   1:  PR[GP1:91,2] = PR[GP1:90,2] + 36.838;
   1:L PR[91] R[100]mm/sec CNT100;
   1:  PR[GP1:91,1] = PR[GP1:90,1] + -37.461;
   1:  PR[GP1:91,2] = PR[GP1:90,2] + 32.882;
   1:L PR[91] R[100]mm/sec CNT100;
   1:  PR[GP1:91,1] = PR[GP1:90,1] + -42.341;
   1:  PR[GP1:91,2] = PR[GP1:90,2] + 27.004;
   1:L PR[91] R[100]mm/sec CNT100;
   1:  PR[GP1:91,1] = PR[GP1:90,1] + -45.904;
   1:  PR[GP1:91,2] = PR[GP1:90,2] + 21.052;
   1:L PR[91] R[100]mm/sec CNT100;
   1:  PR[GP1:91,1] = PR[GP1:90,1] + -48.927;
   1:  PR[GP1:91,2] = PR[GP1:90,2] + 14.203;
   1:L PR[91] R[100]mm/sec CNT100;
   1:  PR[GP1:91,1] = PR[GP1:90,1] + -50.193;
   1:  PR[GP1:91,2] = PR[GP1:90,2] + 7.261;
   1:L PR[91] R[100]mm/sec CNT100;
   1:  PR[GP1:91,1] = PR[GP1:90,1] + -51.214;
   1:  PR[GP1:91,2] = PR[GP1:90,2] + -0.059;
   1:L PR[91] R[100]mm/sec CNT100;
   1:  PR[GP1:91,1] = PR[GP1:90,1] + -49.961;
   1:  PR[GP1:91,2] = PR[GP1:90,2] + -6.907;
   1:L PR[91] R[100]mm/sec CNT100;
   1:  PR[GP1:91,1] = PR[GP1:90,1] + -48.922;
   1:  PR[GP1:91,2] = PR[GP1:90,2] + -14.358;
   1:L PR[91] R[100]mm/sec CNT100;
   1:  PR[GP1:91,1] = PR[GP1:90,1] + -45.904;
   1:  PR[GP1:91,2] = PR[GP1:90,2] + -21.195;
   1:L PR[91] R[100]mm/sec CNT100;
   1:  PR[GP1:91,1] = PR[GP1:90,1] + -42.341;
   1:  PR[GP1:91,2] = PR[GP1:90,2] + -27.147;
   1:L PR[91] R[100]mm/sec CNT100;
   1:  PR[GP1:91,1] = PR[GP1:90,1] + -37.450;
   1:  PR[GP1:91,2] = PR[GP1:90,2] + -33.039;
   1:L PR[91] R[100]mm/sec CNT100;
   1:  PR[GP1:91,1] = PR[GP1:90,1] + -32.224;
   1:  PR[GP1:91,2] = PR[GP1:90,2] + -37.231;
   1:L PR[91] R[100]mm/sec CNT100;
   1:  PR[GP1:91,1] = PR[GP1:90,1] + -26.484;
   1:  PR[GP1:91,2] = PR[GP1:90,2] + -41.295;
   1:L PR[91] R[100]mm/sec CNT100;
   1:  PR[GP1:91,1] = PR[GP1:90,1] + -19.923;
   1:  PR[GP1:91,2] = PR[GP1:90,2] + -43.838;
   1:L PR[91] R[100]mm/sec CNT100;
   1:  PR[GP1:91,1] = PR[GP1:90,1] + -13.684;
   1:  PR[GP1:91,2] = PR[GP1:90,2] + -45.938;
   1:L PR[91] R[100]mm/sec CNT100;
   1:  PR[GP1:91,1] = PR[GP1:90,1] + -6.476;
   1:  PR[GP1:91,2] = PR[GP1:90,2] + -46.831;
   1:L PR[91] R[100]mm/sec CNT100;
   1:  PR[GP1:91,1] = PR[GP1:90,1] + -0.261;
   1:  PR[GP1:91,2] = PR[GP1:90,2] + -46.697;
   1:L PR[91] R[100]mm/sec CNT100;
   1:  PR[GP1:91,1] = PR[GP1:90,1] + 0.472;
   1:  PR[GP1:91,2] = PR[GP1:90,2] + -46.698;
   1:L PR[91] R[100]mm/sec CNT100;
   1:  PR[GP1:91,1] = PR[GP1:90,1] + 6.688;
   1:  PR[GP1:91,2] = PR[GP1:90,2] + -46.831;
   1:L PR[91] R[100]mm/sec CNT100;
   1:  PR[GP1:91,1] = PR[GP1:90,1] + 13.897;
   1:  PR[GP1:91,2] = PR[GP1:90,2] + -45.938;
   1:L PR[91] R[100]mm/sec CNT100;
   1:  PR[GP1:91,1] = PR[GP1:90,1] + 20.136;
   1:  PR[GP1:91,2] = PR[GP1:90,2] + -43.838;
   1:L PR[91] R[100]mm/sec CNT100;
   1:  PR[GP1:91,1] = PR[GP1:90,1] + 26.682;
   1:  PR[GP1:91,2] = PR[GP1:90,2] + -41.301;
   1:L PR[91] R[100]mm/sec CNT100;
   1:  PR[GP1:91,1] = PR[GP1:90,1] + 32.087;
   1:  PR[GP1:91,2] = PR[GP1:90,2] + -36.981;
   1:L PR[91] R[100]mm/sec CNT100;
   1:  PR[GP1:91,1] = PR[GP1:90,1] + 37.676;
   1:  PR[GP1:91,2] = PR[GP1:90,2] + -33.023;
   1:L PR[91] R[100]mm/sec CNT100;
   1:  PR[GP1:91,1] = PR[GP1:90,1] + 42.555;
   1:  PR[GP1:91,2] = PR[GP1:90,2] + -27.145;
   1:L PR[91] R[100]mm/sec CNT100;
   1:  PR[GP1:91,1] = PR[GP1:90,1] + 46.117;
   1:  PR[GP1:91,2] = PR[GP1:90,2] + -21.197;
   1:L PR[91] R[100]mm/sec CNT100;
   1:  PR[GP1:91,1] = PR[GP1:90,1] + 49.141;
   1:  PR[GP1:91,2] = PR[GP1:90,2] + -14.349;
   1:L PR[91] R[100]mm/sec CNT100;
   1:  PR[GP1:91,1] = PR[GP1:90,1] + 50.406;
   1:  PR[GP1:91,2] = PR[GP1:90,2] + -7.404;
   1:L PR[91] R[100]mm/sec CNT100;
   1:  PR[GP1:91,1] = PR[GP1:90,1] + 51.427;
   1:  PR[GP1:91,2] = PR[GP1:90,2] + -0.085;
   1:L PR[91] R[100]mm/sec CNT100;
   1:  PR[GP1:91,1] = PR[GP1:90,1] + 50.175;
   1:  PR[GP1:91,2] = PR[GP1:90,2] + 6.766;
   1:L PR[91] R[100]mm/sec CNT100;
   1:  PR[GP1:91,1] = PR[GP1:90,1] + 49.135;
   1:  PR[GP1:91,2] = PR[GP1:90,2] + 14.217;
   1:L PR[91] R[100]mm/sec CNT100;
   1:  PR[GP1:91,1] = PR[GP1:90,1] + 46.117;
   1:  PR[GP1:91,2] = PR[GP1:90,2] + 21.053;
   1:L PR[91] R[100]mm/sec CNT100;
   1:  PR[GP1:91,1] = PR[GP1:90,1] + 42.555;
   1:  PR[GP1:91,2] = PR[GP1:90,2] + 27.002;
   1:L PR[91] R[100]mm/sec CNT100;
   1:  PR[GP1:91,1] = PR[GP1:90,1] + 37.664;
   1:  PR[GP1:91,2] = PR[GP1:90,2] + 32.894;
   1:L PR[91] R[100]mm/sec CNT100;
   1:  PR[GP1:91,1] = PR[GP1:90,1] + 32.438;
   1:  PR[GP1:91,2] = PR[GP1:90,2] + 37.087;
   1:L PR[91] R[100]mm/sec CNT100;
   1:  PR[GP1:91,1] = PR[GP1:90,1] + 26.697;
   1:  PR[GP1:91,2] = PR[GP1:90,2] + 41.152;
   1:L PR[91] R[100]mm/sec CNT100;
   1:  PR[GP1:91,1] = PR[GP1:90,1] + 20.134;
   1:  PR[GP1:91,2] = PR[GP1:90,2] + 43.695;
   1:L PR[91] R[100]mm/sec CNT100;
   1:  PR[GP1:91,1] = PR[GP1:90,1] + 13.896;
   1:  PR[GP1:91,2] = PR[GP1:90,2] + 45.794;
   1:L PR[91] R[100]mm/sec CNT100;
   1:  PR[GP1:91,1] = PR[GP1:90,1] + 6.686;
   1:  PR[GP1:91,2] = PR[GP1:90,2] + 46.687;
   1:L PR[91] R[100]mm/sec CNT100;
   1:  PR[GP1:91,1] = PR[GP1:90,1] + 0.472;
   1:  PR[GP1:91,2] = PR[GP1:90,2] + 46.554;
   1:L PR[91] R[100]mm/sec CNT100;
   1:  ! -- Layer/Ebene 193 -- !;
   1:  PR[91] = PR[90];
   1:  PR[GP1:91,1] = PR[GP1:90,1] + -0.240;
   1:  PR[GP1:91,2] = PR[GP1:90,2] + 46.709;
   1:  PR[GP1:91,3] = PR[GP1:90,3] + 118.035;
   1:L PR[91] R[100]mm/sec CNT100;
   1:  PR[GP1:91,1] = PR[GP1:90,1] + -6.104;
   1:  PR[GP1:91,2] = PR[GP1:90,2] + 46.835;
   1:L PR[91] R[100]mm/sec CNT100;
   1:  PR[GP1:91,1] = PR[GP1:90,1] + -13.586;
   1:  PR[GP1:91,2] = PR[GP1:90,2] + 45.908;
   1:L PR[91] R[100]mm/sec CNT100;
   1:  PR[GP1:91,1] = PR[GP1:90,1] + -19.471;
   1:  PR[GP1:91,2] = PR[GP1:90,2] + 43.928;
   1:L PR[91] R[100]mm/sec CNT100;
   1:  PR[GP1:91,1] = PR[GP1:90,1] + -26.286;
   1:  PR[GP1:91,2] = PR[GP1:90,2] + 41.286;
   1:L PR[91] R[100]mm/sec CNT100;
   1:  PR[GP1:91,1] = PR[GP1:90,1] + -31.386;
   1:  PR[GP1:91,2] = PR[GP1:90,2] + 37.212;
   1:L PR[91] R[100]mm/sec CNT100;
   1:  PR[GP1:91,1] = PR[GP1:90,1] + -37.220;
   1:  PR[GP1:91,2] = PR[GP1:90,2] + 33.081;
   1:L PR[91] R[100]mm/sec CNT100;
   1:  PR[GP1:91,1] = PR[GP1:90,1] + -42.317;
   1:  PR[GP1:91,2] = PR[GP1:90,2] + 26.942;
   1:L PR[91] R[100]mm/sec CNT100;
   1:  PR[GP1:91,1] = PR[GP1:90,1] + -45.678;
   1:  PR[GP1:91,2] = PR[GP1:90,2] + 21.327;
   1:L PR[91] R[100]mm/sec CNT100;
   1:  PR[GP1:91,1] = PR[GP1:90,1] + -48.842;
   1:  PR[GP1:91,2] = PR[GP1:90,2] + 14.160;
   1:L PR[91] R[100]mm/sec CNT100;
   1:  PR[GP1:91,1] = PR[GP1:90,1] + -50.036;
   1:  PR[GP1:91,2] = PR[GP1:90,2] + 7.611;
   1:L PR[91] R[100]mm/sec CNT100;
   1:  PR[GP1:91,1] = PR[GP1:90,1] + -51.106;
   1:  PR[GP1:91,2] = PR[GP1:90,2] + -0.059;
   1:L PR[91] R[100]mm/sec CNT100;
   1:  PR[GP1:91,1] = PR[GP1:90,1] + -49.924;
   1:  PR[GP1:91,2] = PR[GP1:90,2] + -6.518;
   1:L PR[91] R[100]mm/sec CNT100;
   1:  PR[GP1:91,1] = PR[GP1:90,1] + -48.837;
   1:  PR[GP1:91,2] = PR[GP1:90,2] + -14.315;
   1:L PR[91] R[100]mm/sec CNT100;
   1:  PR[GP1:91,1] = PR[GP1:90,1] + -45.678;
   1:  PR[GP1:91,2] = PR[GP1:90,2] + -21.471;
   1:L PR[91] R[100]mm/sec CNT100;
   1:  PR[GP1:91,1] = PR[GP1:90,1] + -42.317;
   1:  PR[GP1:91,2] = PR[GP1:90,2] + -27.085;
   1:L PR[91] R[100]mm/sec CNT100;
   1:  PR[GP1:91,1] = PR[GP1:90,1] + -37.209;
   1:  PR[GP1:91,2] = PR[GP1:90,2] + -33.238;
   1:L PR[91] R[100]mm/sec CNT100;
   1:  PR[GP1:91,1] = PR[GP1:90,1] + -32.280;
   1:  PR[GP1:91,2] = PR[GP1:90,2] + -37.192;
   1:L PR[91] R[100]mm/sec CNT100;
   1:  PR[GP1:91,1] = PR[GP1:90,1] + -26.304;
   1:  PR[GP1:91,2] = PR[GP1:90,2] + -41.423;
   1:L PR[91] R[100]mm/sec CNT100;
   1:  PR[GP1:91,1] = PR[GP1:90,1] + -19.472;
   1:  PR[GP1:91,2] = PR[GP1:90,2] + -44.071;
   1:L PR[91] R[100]mm/sec CNT100;
   1:  PR[GP1:91,1] = PR[GP1:90,1] + -13.588;
   1:  PR[GP1:91,2] = PR[GP1:90,2] + -46.052;
   1:L PR[91] R[100]mm/sec CNT100;
   1:  PR[GP1:91,1] = PR[GP1:90,1] + -6.105;
   1:  PR[GP1:91,2] = PR[GP1:90,2] + -46.979;
   1:L PR[91] R[100]mm/sec CNT100;
   1:  PR[GP1:91,1] = PR[GP1:90,1] + -0.241;
   1:  PR[GP1:91,2] = PR[GP1:90,2] + -46.853;
   1:L PR[91] R[100]mm/sec CNT100;
   1:  PR[GP1:91,1] = PR[GP1:90,1] + 0.452;
   1:L PR[91] R[100]mm/sec CNT100;
   1:  PR[GP1:91,1] = PR[GP1:90,1] + 6.317;
   1:  PR[GP1:91,2] = PR[GP1:90,2] + -46.979;
   1:L PR[91] R[100]mm/sec CNT100;
   1:  PR[GP1:91,1] = PR[GP1:90,1] + 13.801;
   1:  PR[GP1:91,2] = PR[GP1:90,2] + -46.052;
   1:L PR[91] R[100]mm/sec CNT100;
   1:  PR[GP1:91,1] = PR[GP1:90,1] + 19.685;
   1:  PR[GP1:91,2] = PR[GP1:90,2] + -44.071;
   1:L PR[91] R[100]mm/sec CNT100;
   1:  PR[GP1:91,1] = PR[GP1:90,1] + 26.501;
   1:  PR[GP1:91,2] = PR[GP1:90,2] + -41.430;
   1:L PR[91] R[100]mm/sec CNT100;
   1:  PR[GP1:91,1] = PR[GP1:90,1] + 31.600;
   1:  PR[GP1:91,2] = PR[GP1:90,2] + -37.354;
   1:L PR[91] R[100]mm/sec CNT100;
   1:  PR[GP1:91,1] = PR[GP1:90,1] + 37.436;
   1:  PR[GP1:91,2] = PR[GP1:90,2] + -33.222;
   1:L PR[91] R[100]mm/sec CNT100;
   1:  PR[GP1:91,1] = PR[GP1:90,1] + 42.531;
   1:  PR[GP1:91,2] = PR[GP1:90,2] + -27.083;
   1:L PR[91] R[100]mm/sec CNT100;
   1:  PR[GP1:91,1] = PR[GP1:90,1] + 45.891;
   1:  PR[GP1:91,2] = PR[GP1:90,2] + -21.472;
   1:L PR[91] R[100]mm/sec CNT100;
   1:  PR[GP1:91,1] = PR[GP1:90,1] + 49.055;
   1:  PR[GP1:91,2] = PR[GP1:90,2] + -14.305;
   1:L PR[91] R[100]mm/sec CNT100;
   1:  PR[GP1:91,1] = PR[GP1:90,1] + 50.249;
   1:  PR[GP1:91,2] = PR[GP1:90,2] + -7.755;
   1:L PR[91] R[100]mm/sec CNT100;
   1:  PR[GP1:91,1] = PR[GP1:90,1] + 51.319;
   1:  PR[GP1:91,2] = PR[GP1:90,2] + -0.085;
   1:L PR[91] R[100]mm/sec CNT100;
   1:  PR[GP1:91,1] = PR[GP1:90,1] + 50.137;
   1:  PR[GP1:91,2] = PR[GP1:90,2] + 6.377;
   1:L PR[91] R[100]mm/sec CNT100;
   1:  PR[GP1:91,1] = PR[GP1:90,1] + 49.050;
   1:  PR[GP1:91,2] = PR[GP1:90,2] + 14.174;
   1:L PR[91] R[100]mm/sec CNT100;
   1:  PR[GP1:91,1] = PR[GP1:90,1] + 45.891;
   1:  PR[GP1:91,2] = PR[GP1:90,2] + 21.329;
   1:L PR[91] R[100]mm/sec CNT100;
   1:  PR[GP1:91,1] = PR[GP1:90,1] + 42.531;
   1:  PR[GP1:91,2] = PR[GP1:90,2] + 26.940;
   1:L PR[91] R[100]mm/sec CNT100;
   1:  PR[GP1:91,1] = PR[GP1:90,1] + 37.423;
   1:  PR[GP1:91,2] = PR[GP1:90,2] + 33.092;
   1:L PR[91] R[100]mm/sec CNT100;
   1:  PR[GP1:91,1] = PR[GP1:90,1] + 32.494;
   1:  PR[GP1:91,2] = PR[GP1:90,2] + 37.048;
   1:L PR[91] R[100]mm/sec CNT100;
   1:  PR[GP1:91,1] = PR[GP1:90,1] + 26.517;
   1:  PR[GP1:91,2] = PR[GP1:90,2] + 41.280;
   1:L PR[91] R[100]mm/sec CNT100;
   1:  PR[GP1:91,1] = PR[GP1:90,1] + 19.684;
   1:  PR[GP1:91,2] = PR[GP1:90,2] + 43.928;
   1:L PR[91] R[100]mm/sec CNT100;
   1:  PR[GP1:91,1] = PR[GP1:90,1] + 13.799;
   1:  PR[GP1:91,2] = PR[GP1:90,2] + 45.908;
   1:L PR[91] R[100]mm/sec CNT100;
   1:  PR[GP1:91,1] = PR[GP1:90,1] + 6.315;
   1:  PR[GP1:91,2] = PR[GP1:90,2] + 46.835;
   1:L PR[91] R[100]mm/sec CNT100;
   1:  PR[GP1:91,1] = PR[GP1:90,1] + 0.452;
   1:  PR[GP1:91,2] = PR[GP1:90,2] + 46.709;
   1:L PR[91] R[100]mm/sec CNT100;
   1:  ! -- Layer/Ebene 194 -- !;
   1:  PR[91] = PR[90];
   1:  PR[GP1:91,1] = PR[GP1:90,1] + -0.220;
   1:  PR[GP1:91,2] = PR[GP1:90,2] + 46.865;
   1:  PR[GP1:91,3] = PR[GP1:90,3] + 118.645;
   1:L PR[91] R[100]mm/sec CNT100;
   1:  PR[GP1:91,1] = PR[GP1:90,1] + -5.733;
   1:  PR[GP1:91,2] = PR[GP1:90,2] + 46.983;
   1:L PR[91] R[100]mm/sec CNT100;
   1:  PR[GP1:91,1] = PR[GP1:90,1] + -13.490;
   1:  PR[GP1:91,2] = PR[GP1:90,2] + 46.022;
   1:L PR[91] R[100]mm/sec CNT100;
   1:  PR[GP1:91,1] = PR[GP1:90,1] + -19.021;
   1:  PR[GP1:91,2] = PR[GP1:90,2] + 44.161;
   1:L PR[91] R[100]mm/sec CNT100;
   1:  PR[GP1:91,1] = PR[GP1:90,1] + -26.106;
   1:  PR[GP1:91,2] = PR[GP1:90,2] + 41.415;
   1:L PR[91] R[100]mm/sec CNT100;
   1:  PR[GP1:91,1] = PR[GP1:90,1] + -30.900;
   1:  PR[GP1:91,2] = PR[GP1:90,2] + 37.585;
   1:L PR[91] R[100]mm/sec CNT100;
   1:  PR[GP1:91,1] = PR[GP1:90,1] + -36.980;
   1:  PR[GP1:91,2] = PR[GP1:90,2] + 33.280;
   1:L PR[91] R[100]mm/sec CNT100;
   1:  PR[GP1:91,1] = PR[GP1:90,1] + -42.293;
   1:  PR[GP1:91,2] = PR[GP1:90,2] + 26.880;
   1:L PR[91] R[100]mm/sec CNT100;
   1:  PR[GP1:91,1] = PR[GP1:90,1] + -45.452;
   1:  PR[GP1:91,2] = PR[GP1:90,2] + 21.603;
   1:L PR[91] R[100]mm/sec CNT100;
   1:  PR[GP1:91,1] = PR[GP1:90,1] + -48.757;
   1:  PR[GP1:91,2] = PR[GP1:90,2] + 14.117;
   1:L PR[91] R[100]mm/sec CNT100;
   1:  PR[GP1:91,1] = PR[GP1:90,1] + -49.879;
   1:  PR[GP1:91,2] = PR[GP1:90,2] + 7.962;
   1:L PR[91] R[100]mm/sec CNT100;
   1:  PR[GP1:91,1] = PR[GP1:90,1] + -50.998;
   1:  PR[GP1:91,2] = PR[GP1:90,2] + -0.059;
   1:L PR[91] R[100]mm/sec CNT100;
   1:  PR[GP1:91,1] = PR[GP1:90,1] + -49.887;
   1:  PR[GP1:91,2] = PR[GP1:90,2] + -6.130;
   1:L PR[91] R[100]mm/sec CNT100;
   1:  PR[GP1:91,1] = PR[GP1:90,1] + -48.752;
   1:  PR[GP1:91,2] = PR[GP1:90,2] + -14.272;
   1:L PR[91] R[100]mm/sec CNT100;
   1:  PR[GP1:91,1] = PR[GP1:90,1] + -45.452;
   1:  PR[GP1:91,2] = PR[GP1:90,2] + -21.747;
   1:L PR[91] R[100]mm/sec CNT100;
   1:  PR[GP1:91,1] = PR[GP1:90,1] + -42.294;
   1:  PR[GP1:91,2] = PR[GP1:90,2] + -27.023;
   1:L PR[91] R[100]mm/sec CNT100;
   1:  PR[GP1:91,1] = PR[GP1:90,1] + -36.969;
   1:  PR[GP1:91,2] = PR[GP1:90,2] + -33.437;
   1:L PR[91] R[100]mm/sec CNT100;
   1:  PR[GP1:91,1] = PR[GP1:90,1] + -32.336;
   1:  PR[GP1:91,2] = PR[GP1:90,2] + -37.153;
   1:L PR[91] R[100]mm/sec CNT100;
   1:  PR[GP1:91,1] = PR[GP1:90,1] + -26.124;
   1:  PR[GP1:91,2] = PR[GP1:90,2] + -41.552;
   1:L PR[91] R[100]mm/sec CNT100;
   1:  PR[GP1:91,1] = PR[GP1:90,1] + -19.022;
   1:  PR[GP1:91,2] = PR[GP1:90,2] + -44.304;
   1:L PR[91] R[100]mm/sec CNT100;
   1:  PR[GP1:91,1] = PR[GP1:90,1] + -13.491;
   1:  PR[GP1:91,2] = PR[GP1:90,2] + -46.166;
   1:L PR[91] R[100]mm/sec CNT100;
   1:  PR[GP1:91,1] = PR[GP1:90,1] + -5.734;
   1:  PR[GP1:91,2] = PR[GP1:90,2] + -47.127;
   1:L PR[91] R[100]mm/sec CNT100;
   1:  PR[GP1:91,1] = PR[GP1:90,1] + -0.221;
   1:  PR[GP1:91,2] = PR[GP1:90,2] + -47.009;
   1:L PR[91] R[100]mm/sec CNT100;
   1:  PR[GP1:91,1] = PR[GP1:90,1] + 0.432;
   1:L PR[91] R[100]mm/sec CNT100;
   1:  PR[GP1:91,1] = PR[GP1:90,1] + 5.946;
   1:  PR[GP1:91,2] = PR[GP1:90,2] + -47.127;
   1:L PR[91] R[100]mm/sec CNT100;
   1:  PR[GP1:91,1] = PR[GP1:90,1] + 13.704;
   1:  PR[GP1:91,2] = PR[GP1:90,2] + -46.166;
   1:L PR[91] R[100]mm/sec CNT100;
   1:  PR[GP1:91,1] = PR[GP1:90,1] + 19.235;
   1:  PR[GP1:91,2] = PR[GP1:90,2] + -44.304;
   1:L PR[91] R[100]mm/sec CNT100;
   1:  PR[GP1:91,1] = PR[GP1:90,1] + 26.321;
   1:  PR[GP1:91,2] = PR[GP1:90,2] + -41.558;
   1:L PR[91] R[100]mm/sec CNT100;
   1:  PR[GP1:91,1] = PR[GP1:90,1] + 31.114;
   1:  PR[GP1:91,2] = PR[GP1:90,2] + -37.727;
   1:L PR[91] R[100]mm/sec CNT100;
   1:  PR[GP1:91,1] = PR[GP1:90,1] + 37.195;
   1:  PR[GP1:91,2] = PR[GP1:90,2] + -33.421;
   1:L PR[91] R[100]mm/sec CNT100;
   1:  PR[GP1:91,1] = PR[GP1:90,1] + 42.507;
   1:  PR[GP1:91,2] = PR[GP1:90,2] + -27.022;
   1:L PR[91] R[100]mm/sec CNT100;
   1:  PR[GP1:91,1] = PR[GP1:90,1] + 45.665;
   1:  PR[GP1:91,2] = PR[GP1:90,2] + -21.748;
   1:L PR[91] R[100]mm/sec CNT100;
   1:  PR[GP1:91,1] = PR[GP1:90,1] + 48.970;
   1:  PR[GP1:91,2] = PR[GP1:90,2] + -14.262;
   1:L PR[91] R[100]mm/sec CNT100;
   1:  PR[GP1:91,1] = PR[GP1:90,1] + 50.092;
   1:  PR[GP1:91,2] = PR[GP1:90,2] + -8.106;
   1:L PR[91] R[100]mm/sec CNT100;
   1:  PR[GP1:91,1] = PR[GP1:90,1] + 51.211;
   1:  PR[GP1:91,2] = PR[GP1:90,2] + -0.085;
   1:L PR[91] R[100]mm/sec CNT100;
   1:  PR[GP1:91,1] = PR[GP1:90,1] + 50.100;
   1:  PR[GP1:91,2] = PR[GP1:90,2] + 5.988;
   1:L PR[91] R[100]mm/sec CNT100;
   1:  PR[GP1:91,1] = PR[GP1:90,1] + 48.965;
   1:  PR[GP1:91,2] = PR[GP1:90,2] + 14.130;
   1:L PR[91] R[100]mm/sec CNT100;
   1:  PR[GP1:91,1] = PR[GP1:90,1] + 45.665;
   1:  PR[GP1:91,2] = PR[GP1:90,2] + 21.604;
   1:L PR[91] R[100]mm/sec CNT100;
   1:  PR[GP1:91,1] = PR[GP1:90,1] + 42.507;
   1:  PR[GP1:91,2] = PR[GP1:90,2] + 26.878;
   1:L PR[91] R[100]mm/sec CNT100;
   1:  PR[GP1:91,1] = PR[GP1:90,1] + 37.183;
   1:  PR[GP1:91,2] = PR[GP1:90,2] + 33.291;
   1:L PR[91] R[100]mm/sec CNT100;
   1:  PR[GP1:91,1] = PR[GP1:90,1] + 32.550;
   1:  PR[GP1:91,2] = PR[GP1:90,2] + 37.009;
   1:L PR[91] R[100]mm/sec CNT100;
   1:  PR[GP1:91,1] = PR[GP1:90,1] + 26.336;
   1:  PR[GP1:91,2] = PR[GP1:90,2] + 41.408;
   1:L PR[91] R[100]mm/sec CNT100;
   1:  PR[GP1:91,1] = PR[GP1:90,1] + 19.234;
   1:  PR[GP1:91,2] = PR[GP1:90,2] + 44.161;
   1:L PR[91] R[100]mm/sec CNT100;
   1:  PR[GP1:91,1] = PR[GP1:90,1] + 13.702;
   1:  PR[GP1:91,2] = PR[GP1:90,2] + 46.023;
   1:L PR[91] R[100]mm/sec CNT100;
   1:  PR[GP1:91,1] = PR[GP1:90,1] + 5.945;
   1:  PR[GP1:91,2] = PR[GP1:90,2] + 46.983;
   1:L PR[91] R[100]mm/sec CNT100;
   1:  PR[GP1:91,1] = PR[GP1:90,1] + 0.432;
   1:  PR[GP1:91,2] = PR[GP1:90,2] + 46.865;
   1:L PR[91] R[100]mm/sec CNT100;
   1:  ! -- Layer/Ebene 195 -- !;
   1:  PR[91] = PR[90];
   1:  PR[GP1:91,1] = PR[GP1:90,1] + -0.200;
   1:  PR[GP1:91,2] = PR[GP1:90,2] + 47.020;
   1:  PR[GP1:91,3] = PR[GP1:90,3] + 119.255;
   1:L PR[91] R[100]mm/sec CNT100;
   1:  PR[GP1:91,1] = PR[GP1:90,1] + -5.362;
   1:  PR[GP1:91,2] = PR[GP1:90,2] + 47.131;
   1:L PR[91] R[100]mm/sec CNT100;
   1:  PR[GP1:91,1] = PR[GP1:90,1] + -13.393;
   1:  PR[GP1:91,2] = PR[GP1:90,2] + 46.136;
   1:L PR[91] R[100]mm/sec CNT100;
   1:  PR[GP1:91,1] = PR[GP1:90,1] + -18.571;
   1:  PR[GP1:91,2] = PR[GP1:90,2] + 44.394;
   1:L PR[91] R[100]mm/sec CNT100;
   1:  PR[GP1:91,1] = PR[GP1:90,1] + -25.926;
   1:  PR[GP1:91,2] = PR[GP1:90,2] + 41.543;
   1:L PR[91] R[100]mm/sec CNT100;
   1:  PR[GP1:91,1] = PR[GP1:90,1] + -30.413;
   1:  PR[GP1:91,2] = PR[GP1:90,2] + 37.958;
   1:L PR[91] R[100]mm/sec CNT100;
   1:  PR[GP1:91,1] = PR[GP1:90,1] + -36.739;
   1:  PR[GP1:91,2] = PR[GP1:90,2] + 33.479;
   1:L PR[91] R[100]mm/sec CNT100;
   1:  PR[GP1:91,1] = PR[GP1:90,1] + -42.269;
   1:  PR[GP1:91,2] = PR[GP1:90,2] + 26.818;
   1:L PR[91] R[100]mm/sec CNT100;
   1:  PR[GP1:91,1] = PR[GP1:90,1] + -45.226;
   1:  PR[GP1:91,2] = PR[GP1:90,2] + 21.879;
   1:L PR[91] R[100]mm/sec CNT100;
   1:  PR[GP1:91,1] = PR[GP1:90,1] + -48.671;
   1:  PR[GP1:91,2] = PR[GP1:90,2] + 14.074;
   1:L PR[91] R[100]mm/sec CNT100;
   1:  PR[GP1:91,1] = PR[GP1:90,1] + -49.722;
   1:  PR[GP1:91,2] = PR[GP1:90,2] + 8.313;
   1:L PR[91] R[100]mm/sec CNT100;
   1:  PR[GP1:91,1] = PR[GP1:90,1] + -50.889;
   1:  PR[GP1:91,2] = PR[GP1:90,2] + -0.059;
   1:L PR[91] R[100]mm/sec CNT100;
   1:  PR[GP1:91,1] = PR[GP1:90,1] + -49.850;
   1:  PR[GP1:91,2] = PR[GP1:90,2] + -5.741;
   1:L PR[91] R[100]mm/sec CNT100;
   1:  PR[GP1:91,1] = PR[GP1:90,1] + -48.666;
   1:  PR[GP1:91,2] = PR[GP1:90,2] + -14.229;
   1:L PR[91] R[100]mm/sec CNT100;
   1:  PR[GP1:91,1] = PR[GP1:90,1] + -45.226;
   1:  PR[GP1:91,2] = PR[GP1:90,2] + -22.022;
   1:L PR[91] R[100]mm/sec CNT100;
   1:  PR[GP1:91,1] = PR[GP1:90,1] + -42.270;
   1:  PR[GP1:91,2] = PR[GP1:90,2] + -26.961;
   1:L PR[91] R[100]mm/sec CNT100;
   1:  PR[GP1:91,1] = PR[GP1:90,1] + -36.728;
   1:  PR[GP1:91,2] = PR[GP1:90,2] + -33.636;
   1:L PR[91] R[100]mm/sec CNT100;
   1:  PR[GP1:91,1] = PR[GP1:90,1] + -32.392;
   1:  PR[GP1:91,2] = PR[GP1:90,2] + -37.114;
   1:L PR[91] R[100]mm/sec CNT100;
   1:  PR[GP1:91,1] = PR[GP1:90,1] + -25.943;
   1:  PR[GP1:91,2] = PR[GP1:90,2] + -41.680;
   1:L PR[91] R[100]mm/sec CNT100;
   1:  PR[GP1:91,1] = PR[GP1:90,1] + -18.572;
   1:  PR[GP1:91,2] = PR[GP1:90,2] + -44.537;
   1:L PR[91] R[100]mm/sec CNT100;
   1:  PR[GP1:91,1] = PR[GP1:90,1] + -13.394;
   1:  PR[GP1:91,2] = PR[GP1:90,2] + -46.280;
   1:L PR[91] R[100]mm/sec CNT100;
   1:  PR[GP1:91,1] = PR[GP1:90,1] + -5.364;
   1:  PR[GP1:91,2] = PR[GP1:90,2] + -47.275;
   1:L PR[91] R[100]mm/sec CNT100;
   1:  PR[GP1:91,1] = PR[GP1:90,1] + -0.201;
   1:  PR[GP1:91,2] = PR[GP1:90,2] + -47.164;
   1:L PR[91] R[100]mm/sec CNT100;
   1:  PR[GP1:91,1] = PR[GP1:90,1] + 0.412;
   1:L PR[91] R[100]mm/sec CNT100;
   1:  PR[GP1:91,1] = PR[GP1:90,1] + 5.575;
   1:  PR[GP1:91,2] = PR[GP1:90,2] + -47.275;
   1:L PR[91] R[100]mm/sec CNT100;
   1:  PR[GP1:91,1] = PR[GP1:90,1] + 13.607;
   1:  PR[GP1:91,2] = PR[GP1:90,2] + -46.280;
   1:L PR[91] R[100]mm/sec CNT100;
   1:  PR[GP1:91,1] = PR[GP1:90,1] + 18.784;
   1:  PR[GP1:91,2] = PR[GP1:90,2] + -44.537;
   1:L PR[91] R[100]mm/sec CNT100;
   1:  PR[GP1:91,1] = PR[GP1:90,1] + 26.140;
   1:  PR[GP1:91,2] = PR[GP1:90,2] + -41.687;
   1:L PR[91] R[100]mm/sec CNT100;
   1:  PR[GP1:91,1] = PR[GP1:90,1] + 30.627;
   1:  PR[GP1:91,2] = PR[GP1:90,2] + -38.101;
   1:L PR[91] R[100]mm/sec CNT100;
   1:  PR[GP1:91,1] = PR[GP1:90,1] + 36.955;
   1:  PR[GP1:91,2] = PR[GP1:90,2] + -33.620;
   1:L PR[91] R[100]mm/sec CNT100;
   1:  PR[GP1:91,1] = PR[GP1:90,1] + 42.484;
   1:  PR[GP1:91,2] = PR[GP1:90,2] + -26.960;
   1:L PR[91] R[100]mm/sec CNT100;
   1:  PR[GP1:91,1] = PR[GP1:90,1] + 45.439;
   1:  PR[GP1:91,2] = PR[GP1:90,2] + -22.024;
   1:L PR[91] R[100]mm/sec CNT100;
   1:  PR[GP1:91,1] = PR[GP1:90,1] + 48.885;
   1:  PR[GP1:91,2] = PR[GP1:90,2] + -14.219;
   1:L PR[91] R[100]mm/sec CNT100;
   1:  PR[GP1:91,1] = PR[GP1:90,1] + 49.935;
   1:  PR[GP1:91,2] = PR[GP1:90,2] + -8.456;
   1:L PR[91] R[100]mm/sec CNT100;
   1:  PR[GP1:91,1] = PR[GP1:90,1] + 51.103;
   1:  PR[GP1:91,2] = PR[GP1:90,2] + -0.085;
   1:L PR[91] R[100]mm/sec CNT100;
   1:  PR[GP1:91,1] = PR[GP1:90,1] + 50.063;
   1:  PR[GP1:91,2] = PR[GP1:90,2] + 5.599;
   1:L PR[91] R[100]mm/sec CNT100;
   1:  PR[GP1:91,1] = PR[GP1:90,1] + 48.880;
   1:  PR[GP1:91,2] = PR[GP1:90,2] + 14.087;
   1:L PR[91] R[100]mm/sec CNT100;
   1:  PR[GP1:91,1] = PR[GP1:90,1] + 45.439;
   1:  PR[GP1:91,2] = PR[GP1:90,2] + 21.880;
   1:L PR[91] R[100]mm/sec CNT100;
   1:  PR[GP1:91,1] = PR[GP1:90,1] + 42.483;
   1:  PR[GP1:91,2] = PR[GP1:90,2] + 26.816;
   1:L PR[91] R[100]mm/sec CNT100;
   1:  PR[GP1:91,1] = PR[GP1:90,1] + 36.943;
   1:  PR[GP1:91,2] = PR[GP1:90,2] + 33.490;
   1:L PR[91] R[100]mm/sec CNT100;
   1:  PR[GP1:91,1] = PR[GP1:90,1] + 32.606;
   1:  PR[GP1:91,2] = PR[GP1:90,2] + 36.970;
   1:L PR[91] R[100]mm/sec CNT100;
   1:  PR[GP1:91,1] = PR[GP1:90,1] + 26.156;
   1:  PR[GP1:91,2] = PR[GP1:90,2] + 41.537;
   1:L PR[91] R[100]mm/sec CNT100;
   1:  PR[GP1:91,1] = PR[GP1:90,1] + 18.783;
   1:  PR[GP1:91,2] = PR[GP1:90,2] + 44.394;
   1:L PR[91] R[100]mm/sec CNT100;
   1:  PR[GP1:91,1] = PR[GP1:90,1] + 13.606;
   1:  PR[GP1:91,2] = PR[GP1:90,2] + 46.137;
   1:L PR[91] R[100]mm/sec CNT100;
   1:  PR[GP1:91,1] = PR[GP1:90,1] + 5.574;
   1:  PR[GP1:91,2] = PR[GP1:90,2] + 47.131;
   1:L PR[91] R[100]mm/sec CNT100;
   1:  PR[GP1:91,1] = PR[GP1:90,1] + 0.411;
   1:  PR[GP1:91,2] = PR[GP1:90,2] + 47.020;
   1:L PR[91] R[100]mm/sec CNT100;
   1:  ! -- Layer/Ebene 196 -- !;
   1:  PR[91] = PR[90];
   1:  PR[GP1:91,1] = PR[GP1:90,1] + -0.180;
   1:  PR[GP1:91,2] = PR[GP1:90,2] + 47.176;
   1:  PR[GP1:91,3] = PR[GP1:90,3] + 119.865;
   1:L PR[91] R[100]mm/sec CNT100;
   1:  PR[GP1:91,1] = PR[GP1:90,1] + -4.992;
   1:  PR[GP1:91,2] = PR[GP1:90,2] + 47.279;
   1:L PR[91] R[100]mm/sec CNT100;
   1:  PR[GP1:91,1] = PR[GP1:90,1] + -13.297;
   1:  PR[GP1:91,2] = PR[GP1:90,2] + 46.250;
   1:L PR[91] R[100]mm/sec CNT100;
   1:  PR[GP1:91,1] = PR[GP1:90,1] + -18.120;
   1:  PR[GP1:91,2] = PR[GP1:90,2] + 44.627;
   1:L PR[91] R[100]mm/sec CNT100;
   1:  PR[GP1:91,1] = PR[GP1:90,1] + -25.746;
   1:  PR[GP1:91,2] = PR[GP1:90,2] + 41.672;
   1:L PR[91] R[100]mm/sec CNT100;
   1:  PR[GP1:91,1] = PR[GP1:90,1] + -29.926;
   1:  PR[GP1:91,2] = PR[GP1:90,2] + 38.331;
   1:L PR[91] R[100]mm/sec CNT100;
   1:  PR[GP1:91,1] = PR[GP1:90,1] + -36.499;
   1:  PR[GP1:91,2] = PR[GP1:90,2] + 33.677;
   1:L PR[91] R[100]mm/sec CNT100;
   1:  PR[GP1:91,1] = PR[GP1:90,1] + -42.245;
   1:  PR[GP1:91,2] = PR[GP1:90,2] + 26.756;
   1:L PR[91] R[100]mm/sec CNT100;
   1:  PR[GP1:91,1] = PR[GP1:90,1] + -45.000;
   1:  PR[GP1:91,2] = PR[GP1:90,2] + 22.155;
   1:L PR[91] R[100]mm/sec CNT100;
   1:  PR[GP1:91,1] = PR[GP1:90,1] + -48.586;
   1:  PR[GP1:91,2] = PR[GP1:90,2] + 14.030;
   1:L PR[91] R[100]mm/sec CNT100;
   1:  PR[GP1:91,1] = PR[GP1:90,1] + -49.565;
   1:  PR[GP1:91,2] = PR[GP1:90,2] + 8.663;
   1:L PR[91] R[100]mm/sec CNT100;
   1:  PR[GP1:91,1] = PR[GP1:90,1] + -50.781;
   1:  PR[GP1:91,2] = PR[GP1:90,2] + -0.059;
   1:L PR[91] R[100]mm/sec CNT100;
   1:  PR[GP1:91,1] = PR[GP1:90,1] + -49.813;
   1:  PR[GP1:91,2] = PR[GP1:90,2] + -5.353;
   1:L PR[91] R[100]mm/sec CNT100;
   1:  PR[GP1:91,1] = PR[GP1:90,1] + -48.581;
   1:  PR[GP1:91,2] = PR[GP1:90,2] + -14.186;
   1:L PR[91] R[100]mm/sec CNT100;
   1:  PR[GP1:91,1] = PR[GP1:90,1] + -45.000;
   1:  PR[GP1:91,2] = PR[GP1:90,2] + -22.298;
   1:L PR[91] R[100]mm/sec CNT100;
   1:  PR[GP1:91,1] = PR[GP1:90,1] + -42.246;
   1:  PR[GP1:91,2] = PR[GP1:90,2] + -26.899;
   1:L PR[91] R[100]mm/sec CNT100;
   1:  PR[GP1:91,1] = PR[GP1:90,1] + -36.488;
   1:  PR[GP1:91,2] = PR[GP1:90,2] + -33.835;
   1:L PR[91] R[100]mm/sec CNT100;
   1:  PR[GP1:91,1] = PR[GP1:90,1] + -32.448;
   1:  PR[GP1:91,2] = PR[GP1:90,2] + -37.075;
   1:L PR[91] R[100]mm/sec CNT100;
   1:  PR[GP1:91,1] = PR[GP1:90,1] + -25.763;
   1:  PR[GP1:91,2] = PR[GP1:90,2] + -41.809;
   1:L PR[91] R[100]mm/sec CNT100;
   1:  PR[GP1:91,1] = PR[GP1:90,1] + -18.121;
   1:  PR[GP1:91,2] = PR[GP1:90,2] + -44.770;
   1:L PR[91] R[100]mm/sec CNT100;
   1:  PR[GP1:91,1] = PR[GP1:90,1] + -13.298;
   1:  PR[GP1:91,2] = PR[GP1:90,2] + -46.394;
   1:L PR[91] R[100]mm/sec CNT100;
   1:  PR[GP1:91,1] = PR[GP1:90,1] + -4.993;
   1:  PR[GP1:91,2] = PR[GP1:90,2] + -47.423;
   1:L PR[91] R[100]mm/sec CNT100;
   1:  PR[GP1:91,1] = PR[GP1:90,1] + -0.180;
   1:  PR[GP1:91,2] = PR[GP1:90,2] + -47.320;
   1:L PR[91] R[100]mm/sec CNT100;
   1:  PR[GP1:91,1] = PR[GP1:90,1] + 0.391;
   1:L PR[91] R[100]mm/sec CNT100;
   1:  PR[GP1:91,1] = PR[GP1:90,1] + 5.204;
   1:  PR[GP1:91,2] = PR[GP1:90,2] + -47.423;
   1:L PR[91] R[100]mm/sec CNT100;
   1:  PR[GP1:91,1] = PR[GP1:90,1] + 13.510;
   1:  PR[GP1:91,2] = PR[GP1:90,2] + -46.395;
   1:L PR[91] R[100]mm/sec CNT100;
   1:  PR[GP1:91,1] = PR[GP1:90,1] + 18.334;
   1:  PR[GP1:91,2] = PR[GP1:90,2] + -44.771;
   1:L PR[91] R[100]mm/sec CNT100;
   1:  PR[GP1:91,1] = PR[GP1:90,1] + 25.960;
   1:  PR[GP1:91,2] = PR[GP1:90,2] + -41.815;
   1:L PR[91] R[100]mm/sec CNT100;
   1:  PR[GP1:91,1] = PR[GP1:90,1] + 30.140;
   1:  PR[GP1:91,2] = PR[GP1:90,2] + -38.474;
   1:L PR[91] R[100]mm/sec CNT100;
   1:  PR[GP1:91,1] = PR[GP1:90,1] + 36.714;
   1:  PR[GP1:91,2] = PR[GP1:90,2] + -33.819;
   1:L PR[91] R[100]mm/sec CNT100;
   1:  PR[GP1:91,1] = PR[GP1:90,1] + 42.460;
   1:  PR[GP1:91,2] = PR[GP1:90,2] + -26.898;
   1:L PR[91] R[100]mm/sec CNT100;
   1:  PR[GP1:91,1] = PR[GP1:90,1] + 45.213;
   1:  PR[GP1:91,2] = PR[GP1:90,2] + -22.299;
   1:L PR[91] R[100]mm/sec CNT100;
   1:  PR[GP1:91,1] = PR[GP1:90,1] + 48.800;
   1:  PR[GP1:91,2] = PR[GP1:90,2] + -14.175;
   1:L PR[91] R[100]mm/sec CNT100;
   1:  PR[GP1:91,1] = PR[GP1:90,1] + 49.778;
   1:  PR[GP1:91,2] = PR[GP1:90,2] + -8.807;
   1:L PR[91] R[100]mm/sec CNT100;
   1:  PR[GP1:91,1] = PR[GP1:90,1] + 50.995;
   1:  PR[GP1:91,2] = PR[GP1:90,2] + -0.085;
   1:L PR[91] R[100]mm/sec CNT100;
   1:  PR[GP1:91,1] = PR[GP1:90,1] + 50.026;
   1:  PR[GP1:91,2] = PR[GP1:90,2] + 5.211;
   1:L PR[91] R[100]mm/sec CNT100;
   1:  PR[GP1:91,1] = PR[GP1:90,1] + 48.794;
   1:  PR[GP1:91,2] = PR[GP1:90,2] + 14.043;
   1:L PR[91] R[100]mm/sec CNT100;
   1:  PR[GP1:91,1] = PR[GP1:90,1] + 45.213;
   1:  PR[GP1:91,2] = PR[GP1:90,2] + 22.156;
   1:L PR[91] R[100]mm/sec CNT100;
   1:  PR[GP1:91,1] = PR[GP1:90,1] + 42.459;
   1:  PR[GP1:91,2] = PR[GP1:90,2] + 26.754;
   1:L PR[91] R[100]mm/sec CNT100;
   1:  PR[GP1:91,1] = PR[GP1:90,1] + 36.702;
   1:  PR[GP1:91,2] = PR[GP1:90,2] + 33.689;
   1:L PR[91] R[100]mm/sec CNT100;
   1:  PR[GP1:91,1] = PR[GP1:90,1] + 32.662;
   1:  PR[GP1:91,2] = PR[GP1:90,2] + 36.931;
   1:L PR[91] R[100]mm/sec CNT100;
   1:  PR[GP1:91,1] = PR[GP1:90,1] + 25.976;
   1:  PR[GP1:91,2] = PR[GP1:90,2] + 41.665;
   1:L PR[91] R[100]mm/sec CNT100;
   1:  PR[GP1:91,1] = PR[GP1:90,1] + 18.333;
   1:  PR[GP1:91,2] = PR[GP1:90,2] + 44.627;
   1:L PR[91] R[100]mm/sec CNT100;
   1:  PR[GP1:91,1] = PR[GP1:90,1] + 13.509;
   1:  PR[GP1:91,2] = PR[GP1:90,2] + 46.251;
   1:L PR[91] R[100]mm/sec CNT100;
   1:  PR[GP1:91,1] = PR[GP1:90,1] + 5.203;
   1:  PR[GP1:91,2] = PR[GP1:90,2] + 47.279;
   1:L PR[91] R[100]mm/sec CNT100;
   1:  PR[GP1:91,1] = PR[GP1:90,1] + 0.391;
   1:  PR[GP1:91,2] = PR[GP1:90,2] + 47.176;
   1:L PR[91] R[100]mm/sec CNT100;
   1:  ! -- Layer/Ebene 197 -- !;
   1:  PR[91] = PR[90];
   1:  PR[GP1:91,1] = PR[GP1:90,1] + -4.621;
   1:  PR[GP1:91,2] = PR[GP1:90,2] + 47.427;
   1:  PR[GP1:91,3] = PR[GP1:90,3] + 120.475;
   1:L PR[91] R[100]mm/sec CNT100;
   1:  PR[GP1:91,1] = PR[GP1:90,1] + -13.200;
   1:  PR[GP1:91,2] = PR[GP1:90,2] + 46.364;
   1:L PR[91] R[100]mm/sec CNT100;
   1:  PR[GP1:91,1] = PR[GP1:90,1] + -17.670;
   1:  PR[GP1:91,2] = PR[GP1:90,2] + 44.860;
   1:L PR[91] R[100]mm/sec CNT100;
   1:  PR[GP1:91,1] = PR[GP1:90,1] + -25.565;
   1:  PR[GP1:91,2] = PR[GP1:90,2] + 41.800;
   1:L PR[91] R[100]mm/sec CNT100;
   1:  PR[GP1:91,1] = PR[GP1:90,1] + -29.440;
   1:  PR[GP1:91,2] = PR[GP1:90,2] + 38.705;
   1:L PR[91] R[100]mm/sec CNT100;
   1:  PR[GP1:91,1] = PR[GP1:90,1] + -36.259;
   1:  PR[GP1:91,2] = PR[GP1:90,2] + 33.876;
   1:L PR[91] R[100]mm/sec CNT100;
   1:  PR[GP1:91,1] = PR[GP1:90,1] + -42.221;
   1:  PR[GP1:91,2] = PR[GP1:90,2] + 26.694;
   1:L PR[91] R[100]mm/sec CNT100;
   1:  PR[GP1:91,1] = PR[GP1:90,1] + -44.774;
   1:  PR[GP1:91,2] = PR[GP1:90,2] + 22.430;
   1:L PR[91] R[100]mm/sec CNT100;
   1:  PR[GP1:91,1] = PR[GP1:90,1] + -48.501;
   1:  PR[GP1:91,2] = PR[GP1:90,2] + 13.987;
   1:L PR[91] R[100]mm/sec CNT100;
   1:  PR[GP1:91,1] = PR[GP1:90,1] + -49.408;
   1:  PR[GP1:91,2] = PR[GP1:90,2] + 9.014;
   1:L PR[91] R[100]mm/sec CNT100;
   1:  PR[GP1:91,1] = PR[GP1:90,1] + -50.673;
   1:  PR[GP1:91,2] = PR[GP1:90,2] + -0.059;
   1:L PR[91] R[100]mm/sec CNT100;
   1:  PR[GP1:91,1] = PR[GP1:90,1] + -49.776;
   1:  PR[GP1:91,2] = PR[GP1:90,2] + -4.964;
   1:L PR[91] R[100]mm/sec CNT100;
   1:  PR[GP1:91,1] = PR[GP1:90,1] + -48.496;
   1:  PR[GP1:91,2] = PR[GP1:90,2] + -14.142;
   1:L PR[91] R[100]mm/sec CNT100;
   1:  PR[GP1:91,1] = PR[GP1:90,1] + -44.774;
   1:  PR[GP1:91,2] = PR[GP1:90,2] + -22.574;
   1:L PR[91] R[100]mm/sec CNT100;
   1:  PR[GP1:91,1] = PR[GP1:90,1] + -42.222;
   1:  PR[GP1:91,2] = PR[GP1:90,2] + -26.837;
   1:L PR[91] R[100]mm/sec CNT100;
   1:  PR[GP1:91,1] = PR[GP1:90,1] + -36.247;
   1:  PR[GP1:91,2] = PR[GP1:90,2] + -34.034;
   1:L PR[91] R[100]mm/sec CNT100;
   1:  PR[GP1:91,1] = PR[GP1:90,1] + -32.504;
   1:  PR[GP1:91,2] = PR[GP1:90,2] + -37.036;
   1:L PR[91] R[100]mm/sec CNT100;
   1:  PR[GP1:91,1] = PR[GP1:90,1] + -25.583;
   1:  PR[GP1:91,2] = PR[GP1:90,2] + -41.937;
   1:L PR[91] R[100]mm/sec CNT100;
   1:  PR[GP1:91,1] = PR[GP1:90,1] + -17.671;
   1:  PR[GP1:91,2] = PR[GP1:90,2] + -45.004;
   1:L PR[91] R[100]mm/sec CNT100;
   1:  PR[GP1:91,1] = PR[GP1:90,1] + -13.201;
   1:  PR[GP1:91,2] = PR[GP1:90,2] + -46.508;
   1:L PR[91] R[100]mm/sec CNT100;
   1:  PR[GP1:91,1] = PR[GP1:90,1] + -4.623;
   1:  PR[GP1:91,2] = PR[GP1:90,2] + -47.571;
   1:L PR[91] R[100]mm/sec CNT100;
   1:  PR[GP1:91,1] = PR[GP1:90,1] + -0.155;
   1:  PR[GP1:91,2] = PR[GP1:90,2] + -47.475;
   1:L PR[91] R[100]mm/sec CNT100;
   1:  PR[GP1:91,1] = PR[GP1:90,1] + 4.833;
   1:  PR[GP1:91,2] = PR[GP1:90,2] + -47.571;
   1:L PR[91] R[100]mm/sec CNT100;
   1:  PR[GP1:91,1] = PR[GP1:90,1] + 13.413;
   1:  PR[GP1:91,2] = PR[GP1:90,2] + -46.509;
   1:L PR[91] R[100]mm/sec CNT100;
   1:  PR[GP1:91,1] = PR[GP1:90,1] + 17.883;
   1:  PR[GP1:91,2] = PR[GP1:90,2] + -45.004;
   1:L PR[91] R[100]mm/sec CNT100;
   1:  PR[GP1:91,1] = PR[GP1:90,1] + 25.780;
   1:  PR[GP1:91,2] = PR[GP1:90,2] + -41.944;
   1:L PR[91] R[100]mm/sec CNT100;
   1:  PR[GP1:91,1] = PR[GP1:90,1] + 29.653;
   1:  PR[GP1:91,2] = PR[GP1:90,2] + -38.847;
   1:L PR[91] R[100]mm/sec CNT100;
   1:  PR[GP1:91,1] = PR[GP1:90,1] + 36.474;
   1:  PR[GP1:91,2] = PR[GP1:90,2] + -34.018;
   1:L PR[91] R[100]mm/sec CNT100;
   1:  PR[GP1:91,1] = PR[GP1:90,1] + 42.436;
   1:  PR[GP1:91,2] = PR[GP1:90,2] + -26.836;
   1:L PR[91] R[100]mm/sec CNT100;
   1:  PR[GP1:91,1] = PR[GP1:90,1] + 44.987;
   1:  PR[GP1:91,2] = PR[GP1:90,2] + -22.575;
   1:L PR[91] R[100]mm/sec CNT100;
   1:  PR[GP1:91,1] = PR[GP1:90,1] + 48.715;
   1:  PR[GP1:91,2] = PR[GP1:90,2] + -14.132;
   1:L PR[91] R[100]mm/sec CNT100;
   1:  PR[GP1:91,1] = PR[GP1:90,1] + 49.621;
   1:  PR[GP1:91,2] = PR[GP1:90,2] + -9.157;
   1:L PR[91] R[100]mm/sec CNT100;
   1:  PR[GP1:91,1] = PR[GP1:90,1] + 50.887;
   1:  PR[GP1:91,2] = PR[GP1:90,2] + -0.085;
   1:L PR[91] R[100]mm/sec CNT100;
   1:  PR[GP1:91,1] = PR[GP1:90,1] + 49.989;
   1:  PR[GP1:91,2] = PR[GP1:90,2] + 4.822;
   1:L PR[91] R[100]mm/sec CNT100;
   1:  PR[GP1:91,1] = PR[GP1:90,1] + 48.709;
   1:  PR[GP1:91,2] = PR[GP1:90,2] + 14.000;
   1:L PR[91] R[100]mm/sec CNT100;
   1:  PR[GP1:91,1] = PR[GP1:90,1] + 44.987;
   1:  PR[GP1:91,2] = PR[GP1:90,2] + 22.431;
   1:L PR[91] R[100]mm/sec CNT100;
   1:  PR[GP1:91,1] = PR[GP1:90,1] + 42.435;
   1:  PR[GP1:91,2] = PR[GP1:90,2] + 26.692;
   1:L PR[91] R[100]mm/sec CNT100;
   1:  PR[GP1:91,1] = PR[GP1:90,1] + 36.462;
   1:  PR[GP1:91,2] = PR[GP1:90,2] + 33.888;
   1:L PR[91] R[100]mm/sec CNT100;
   1:  PR[GP1:91,1] = PR[GP1:90,1] + 32.718;
   1:  PR[GP1:91,2] = PR[GP1:90,2] + 36.892;
   1:L PR[91] R[100]mm/sec CNT100;
   1:  PR[GP1:91,1] = PR[GP1:90,1] + 25.795;
   1:  PR[GP1:91,2] = PR[GP1:90,2] + 41.794;
   1:L PR[91] R[100]mm/sec CNT100;
   1:  PR[GP1:91,1] = PR[GP1:90,1] + 17.882;
   1:  PR[GP1:91,2] = PR[GP1:90,2] + 44.860;
   1:L PR[91] R[100]mm/sec CNT100;
   1:  PR[GP1:91,1] = PR[GP1:90,1] + 13.412;
   1:  PR[GP1:91,2] = PR[GP1:90,2] + 46.365;
   1:L PR[91] R[100]mm/sec CNT100;
   1:  PR[GP1:91,1] = PR[GP1:90,1] + 4.832;
   1:  PR[GP1:91,2] = PR[GP1:90,2] + 47.427;
   1:L PR[91] R[100]mm/sec CNT100;
   1:  PR[GP1:91,1] = PR[GP1:90,1] + -0.154;
   1:  PR[GP1:91,2] = PR[GP1:90,2] + 47.331;
   1:L PR[91] R[100]mm/sec CNT100;
   1:  ! -- Layer/Ebene 198 -- !;
   1:  PR[91] = PR[90];
   1:  PR[GP1:91,1] = PR[GP1:90,1] + -4.251;
   1:  PR[GP1:91,2] = PR[GP1:90,2] + 47.575;
   1:  PR[GP1:91,3] = PR[GP1:90,3] + 121.085;
   1:L PR[91] R[100]mm/sec CNT100;
   1:  PR[GP1:91,1] = PR[GP1:90,1] + -13.103;
   1:  PR[GP1:91,2] = PR[GP1:90,2] + 46.478;
   1:L PR[91] R[100]mm/sec CNT100;
   1:  PR[GP1:91,1] = PR[GP1:90,1] + -17.220;
   1:  PR[GP1:91,2] = PR[GP1:90,2] + 45.093;
   1:L PR[91] R[100]mm/sec CNT100;
   1:  PR[GP1:91,1] = PR[GP1:90,1] + -25.385;
   1:  PR[GP1:91,2] = PR[GP1:90,2] + 41.929;
   1:L PR[91] R[100]mm/sec CNT100;
   1:  PR[GP1:91,1] = PR[GP1:90,1] + -28.953;
   1:  PR[GP1:91,2] = PR[GP1:90,2] + 39.078;
   1:L PR[91] R[100]mm/sec CNT100;
   1:  PR[GP1:91,1] = PR[GP1:90,1] + -36.018;
   1:  PR[GP1:91,2] = PR[GP1:90,2] + 34.075;
   1:L PR[91] R[100]mm/sec CNT100;
   1:  PR[GP1:91,1] = PR[GP1:90,1] + -42.198;
   1:  PR[GP1:91,2] = PR[GP1:90,2] + 26.632;
   1:L PR[91] R[100]mm/sec CNT100;
   1:  PR[GP1:91,1] = PR[GP1:90,1] + -44.548;
   1:  PR[GP1:91,2] = PR[GP1:90,2] + 22.706;
   1:L PR[91] R[100]mm/sec CNT100;
   1:  PR[GP1:91,1] = PR[GP1:90,1] + -48.416;
   1:  PR[GP1:91,2] = PR[GP1:90,2] + 13.944;
   1:L PR[91] R[100]mm/sec CNT100;
   1:  PR[GP1:91,1] = PR[GP1:90,1] + -49.251;
   1:  PR[GP1:91,2] = PR[GP1:90,2] + 9.364;
   1:L PR[91] R[100]mm/sec CNT100;
   1:  PR[GP1:91,1] = PR[GP1:90,1] + -50.565;
   1:  PR[GP1:91,2] = PR[GP1:90,2] + -0.059;
   1:L PR[91] R[100]mm/sec CNT100;
   1:  PR[GP1:91,1] = PR[GP1:90,1] + -49.739;
   1:  PR[GP1:91,2] = PR[GP1:90,2] + -4.576;
   1:L PR[91] R[100]mm/sec CNT100;
   1:  PR[GP1:91,1] = PR[GP1:90,1] + -48.411;
   1:  PR[GP1:91,2] = PR[GP1:90,2] + -14.099;
   1:L PR[91] R[100]mm/sec CNT100;
   1:  PR[GP1:91,1] = PR[GP1:90,1] + -44.548;
   1:  PR[GP1:91,2] = PR[GP1:90,2] + -22.850;
   1:L PR[91] R[100]mm/sec CNT100;
   1:  PR[GP1:91,1] = PR[GP1:90,1] + -42.198;
   1:  PR[GP1:91,2] = PR[GP1:90,2] + -26.775;
   1:L PR[91] R[100]mm/sec CNT100;
   1:  PR[GP1:91,1] = PR[GP1:90,1] + -36.007;
   1:  PR[GP1:91,2] = PR[GP1:90,2] + -34.233;
   1:L PR[91] R[100]mm/sec CNT100;
   1:  PR[GP1:91,1] = PR[GP1:90,1] + -32.560;
   1:  PR[GP1:91,2] = PR[GP1:90,2] + -36.997;
   1:L PR[91] R[100]mm/sec CNT100;
   1:  PR[GP1:91,1] = PR[GP1:90,1] + -25.402;
   1:  PR[GP1:91,2] = PR[GP1:90,2] + -42.066;
   1:L PR[91] R[100]mm/sec CNT100;
   1:  PR[GP1:91,1] = PR[GP1:90,1] + -17.220;
   1:  PR[GP1:91,2] = PR[GP1:90,2] + -45.237;
   1:L PR[91] R[100]mm/sec CNT100;
   1:  PR[GP1:91,1] = PR[GP1:90,1] + -13.104;
   1:  PR[GP1:91,2] = PR[GP1:90,2] + -46.622;
   1:L PR[91] R[100]mm/sec CNT100;
   1:  PR[GP1:91,1] = PR[GP1:90,1] + -4.252;
   1:  PR[GP1:91,2] = PR[GP1:90,2] + -47.719;
   1:L PR[91] R[100]mm/sec CNT100;
   1:  PR[GP1:91,1] = PR[GP1:90,1] + -0.134;
   1:  PR[GP1:91,2] = PR[GP1:90,2] + -47.631;
   1:L PR[91] R[100]mm/sec CNT100;
   1:  PR[GP1:91,1] = PR[GP1:90,1] + 4.462;
   1:  PR[GP1:91,2] = PR[GP1:90,2] + -47.719;
   1:L PR[91] R[100]mm/sec CNT100;
   1:  PR[GP1:91,1] = PR[GP1:90,1] + 13.317;
   1:  PR[GP1:91,2] = PR[GP1:90,2] + -46.623;
   1:L PR[91] R[100]mm/sec CNT100;
   1:  PR[GP1:91,1] = PR[GP1:90,1] + 17.433;
   1:  PR[GP1:91,2] = PR[GP1:90,2] + -45.237;
   1:L PR[91] R[100]mm/sec CNT100;
   1:  PR[GP1:91,1] = PR[GP1:90,1] + 25.599;
   1:  PR[GP1:91,2] = PR[GP1:90,2] + -42.072;
   1:L PR[91] R[100]mm/sec CNT100;
   1:  PR[GP1:91,1] = PR[GP1:90,1] + 29.167;
   1:  PR[GP1:91,2] = PR[GP1:90,2] + -39.221;
   1:L PR[91] R[100]mm/sec CNT100;
   1:  PR[GP1:91,1] = PR[GP1:90,1] + 36.233;
   1:  PR[GP1:91,2] = PR[GP1:90,2] + -34.217;
   1:L PR[91] R[100]mm/sec CNT100;
   1:  PR[GP1:91,1] = PR[GP1:90,1] + 42.412;
   1:  PR[GP1:91,2] = PR[GP1:90,2] + -26.774;
   1:L PR[91] R[100]mm/sec CNT100;
   1:  PR[GP1:91,1] = PR[GP1:90,1] + 44.761;
   1:  PR[GP1:91,2] = PR[GP1:90,2] + -22.850;
   1:L PR[91] R[100]mm/sec CNT100;
   1:  PR[GP1:91,1] = PR[GP1:90,1] + 48.629;
   1:  PR[GP1:91,2] = PR[GP1:90,2] + -14.089;
   1:L PR[91] R[100]mm/sec CNT100;
   1:  PR[GP1:91,1] = PR[GP1:90,1] + 49.464;
   1:  PR[GP1:91,2] = PR[GP1:90,2] + -9.508;
   1:L PR[91] R[100]mm/sec CNT100;
   1:  PR[GP1:91,1] = PR[GP1:90,1] + 50.778;
   1:  PR[GP1:91,2] = PR[GP1:90,2] + -0.085;
   1:L PR[91] R[100]mm/sec CNT100;
   1:  PR[GP1:91,1] = PR[GP1:90,1] + 49.952;
   1:  PR[GP1:91,2] = PR[GP1:90,2] + 4.433;
   1:L PR[91] R[100]mm/sec CNT100;
   1:  PR[GP1:91,1] = PR[GP1:90,1] + 48.624;
   1:  PR[GP1:91,2] = PR[GP1:90,2] + 13.957;
   1:L PR[91] R[100]mm/sec CNT100;
   1:  PR[GP1:91,1] = PR[GP1:90,1] + 44.761;
   1:  PR[GP1:91,2] = PR[GP1:90,2] + 22.707;
   1:L PR[91] R[100]mm/sec CNT100;
   1:  PR[GP1:91,1] = PR[GP1:90,1] + 42.412;
   1:  PR[GP1:91,2] = PR[GP1:90,2] + 26.630;
   1:L PR[91] R[100]mm/sec CNT100;
   1:  PR[GP1:91,1] = PR[GP1:90,1] + 36.221;
   1:  PR[GP1:91,2] = PR[GP1:90,2] + 34.087;
   1:L PR[91] R[100]mm/sec CNT100;
   1:  PR[GP1:91,1] = PR[GP1:90,1] + 32.774;
   1:  PR[GP1:91,2] = PR[GP1:90,2] + 36.853;
   1:L PR[91] R[100]mm/sec CNT100;
   1:  PR[GP1:91,1] = PR[GP1:90,1] + 25.615;
   1:  PR[GP1:91,2] = PR[GP1:90,2] + 41.922;
   1:L PR[91] R[100]mm/sec CNT100;
   1:  PR[GP1:91,1] = PR[GP1:90,1] + 17.432;
   1:  PR[GP1:91,2] = PR[GP1:90,2] + 45.093;
   1:L PR[91] R[100]mm/sec CNT100;
   1:  PR[GP1:91,1] = PR[GP1:90,1] + 13.316;
   1:  PR[GP1:91,2] = PR[GP1:90,2] + 46.479;
   1:L PR[91] R[100]mm/sec CNT100;
   1:  PR[GP1:91,1] = PR[GP1:90,1] + 4.461;
   1:  PR[GP1:91,2] = PR[GP1:90,2] + 47.575;
   1:L PR[91] R[100]mm/sec CNT100;
   1:  PR[GP1:91,1] = PR[GP1:90,1] + -0.134;
   1:  PR[GP1:91,2] = PR[GP1:90,2] + 47.487;
   1:L PR[91] R[100]mm/sec CNT100;
   1:  ! -- Layer/Ebene 199 -- !;
   1:  PR[91] = PR[90];
   1:  PR[GP1:91,1] = PR[GP1:90,1] + -3.880;
   1:  PR[GP1:91,2] = PR[GP1:90,2] + 47.723;
   1:  PR[GP1:91,3] = PR[GP1:90,3] + 121.695;
   1:L PR[91] R[100]mm/sec CNT100;
   1:  PR[GP1:91,1] = PR[GP1:90,1] + -13.007;
   1:  PR[GP1:91,2] = PR[GP1:90,2] + 46.593;
   1:L PR[91] R[100]mm/sec CNT100;
   1:  PR[GP1:91,1] = PR[GP1:90,1] + -16.769;
   1:  PR[GP1:91,2] = PR[GP1:90,2] + 45.326;
   1:L PR[91] R[100]mm/sec CNT100;
   1:  PR[GP1:91,1] = PR[GP1:90,1] + -25.205;
   1:  PR[GP1:91,2] = PR[GP1:90,2] + 42.057;
   1:L PR[91] R[100]mm/sec CNT100;
   1:  PR[GP1:91,1] = PR[GP1:90,1] + -28.466;
   1:  PR[GP1:91,2] = PR[GP1:90,2] + 39.451;
   1:L PR[91] R[100]mm/sec CNT100;
   1:  PR[GP1:91,1] = PR[GP1:90,1] + -35.778;
   1:  PR[GP1:91,2] = PR[GP1:90,2] + 34.274;
   1:L PR[91] R[100]mm/sec CNT100;
   1:  PR[GP1:91,1] = PR[GP1:90,1] + -42.174;
   1:  PR[GP1:91,2] = PR[GP1:90,2] + 26.570;
   1:L PR[91] R[100]mm/sec CNT100;
   1:  PR[GP1:91,1] = PR[GP1:90,1] + -44.322;
   1:  PR[GP1:91,2] = PR[GP1:90,2] + 22.982;
   1:L PR[91] R[100]mm/sec CNT100;
   1:  PR[GP1:91,1] = PR[GP1:90,1] + -48.331;
   1:  PR[GP1:91,2] = PR[GP1:90,2] + 13.901;
   1:L PR[91] R[100]mm/sec CNT100;
   1:  PR[GP1:91,1] = PR[GP1:90,1] + -49.094;
   1:  PR[GP1:91,2] = PR[GP1:90,2] + 9.715;
   1:L PR[91] R[100]mm/sec CNT100;
   1:  PR[GP1:91,1] = PR[GP1:90,1] + -50.457;
   1:  PR[GP1:91,2] = PR[GP1:90,2] + -0.059;
   1:L PR[91] R[100]mm/sec CNT100;
   1:  PR[GP1:91,1] = PR[GP1:90,1] + -49.702;
   1:  PR[GP1:91,2] = PR[GP1:90,2] + -4.187;
   1:L PR[91] R[100]mm/sec CNT100;
   1:  PR[GP1:91,1] = PR[GP1:90,1] + -48.326;
   1:  PR[GP1:91,2] = PR[GP1:90,2] + -14.056;
   1:L PR[91] R[100]mm/sec CNT100;
   1:  PR[GP1:91,1] = PR[GP1:90,1] + -44.322;
   1:  PR[GP1:91,2] = PR[GP1:90,2] + -23.125;
   1:L PR[91] R[100]mm/sec CNT100;
   1:  PR[GP1:91,1] = PR[GP1:90,1] + -42.174;
   1:  PR[GP1:91,2] = PR[GP1:90,2] + -26.714;
   1:L PR[91] R[100]mm/sec CNT100;
   1:  PR[GP1:91,1] = PR[GP1:90,1] + -35.766;
   1:  PR[GP1:91,2] = PR[GP1:90,2] + -34.432;
   1:L PR[91] R[100]mm/sec CNT100;
   1:  PR[GP1:91,1] = PR[GP1:90,1] + -32.616;
   1:  PR[GP1:91,2] = PR[GP1:90,2] + -36.959;
   1:L PR[91] R[100]mm/sec CNT100;
   1:  PR[GP1:91,1] = PR[GP1:90,1] + -25.222;
   1:  PR[GP1:91,2] = PR[GP1:90,2] + -42.194;
   1:L PR[91] R[100]mm/sec CNT100;
   1:  PR[GP1:91,1] = PR[GP1:90,1] + -16.770;
   1:  PR[GP1:91,2] = PR[GP1:90,2] + -45.470;
   1:L PR[91] R[100]mm/sec CNT100;
   1:  PR[GP1:91,1] = PR[GP1:90,1] + -13.008;
   1:  PR[GP1:91,2] = PR[GP1:90,2] + -46.736;
   1:L PR[91] R[100]mm/sec CNT100;
   1:  PR[GP1:91,1] = PR[GP1:90,1] + -3.881;
   1:  PR[GP1:91,2] = PR[GP1:90,2] + -47.867;
   1:L PR[91] R[100]mm/sec CNT100;
   1:  PR[GP1:91,1] = PR[GP1:90,1] + -0.114;
   1:  PR[GP1:91,2] = PR[GP1:90,2] + -47.786;
   1:L PR[91] R[100]mm/sec CNT100;
   1:  PR[GP1:91,1] = PR[GP1:90,1] + 4.091;
   1:  PR[GP1:91,2] = PR[GP1:90,2] + -47.867;
   1:L PR[91] R[100]mm/sec CNT100;
   1:  PR[GP1:91,1] = PR[GP1:90,1] + 13.220;
   1:  PR[GP1:91,2] = PR[GP1:90,2] + -46.737;
   1:L PR[91] R[100]mm/sec CNT100;
   1:  PR[GP1:91,1] = PR[GP1:90,1] + 16.982;
   1:  PR[GP1:91,2] = PR[GP1:90,2] + -45.470;
   1:L PR[91] R[100]mm/sec CNT100;
   1:  PR[GP1:91,1] = PR[GP1:90,1] + 25.419;
   1:  PR[GP1:91,2] = PR[GP1:90,2] + -42.201;
   1:L PR[91] R[100]mm/sec CNT100;
   1:  PR[GP1:91,1] = PR[GP1:90,1] + 28.680;
   1:  PR[GP1:91,2] = PR[GP1:90,2] + -39.594;
   1:L PR[91] R[100]mm/sec CNT100;
   1:  PR[GP1:91,1] = PR[GP1:90,1] + 35.993;
   1:  PR[GP1:91,2] = PR[GP1:90,2] + -34.416;
   1:L PR[91] R[100]mm/sec CNT100;
   1:  PR[GP1:91,1] = PR[GP1:90,1] + 42.388;
   1:  PR[GP1:91,2] = PR[GP1:90,2] + -26.712;
   1:L PR[91] R[100]mm/sec CNT100;
   1:  PR[GP1:91,1] = PR[GP1:90,1] + 44.535;
   1:  PR[GP1:91,2] = PR[GP1:90,2] + -23.126;
   1:L PR[91] R[100]mm/sec CNT100;
   1:  PR[GP1:91,1] = PR[GP1:90,1] + 48.544;
   1:  PR[GP1:91,2] = PR[GP1:90,2] + -14.045;
   1:L PR[91] R[100]mm/sec CNT100;
   1:  PR[GP1:91,1] = PR[GP1:90,1] + 49.307;
   1:  PR[GP1:91,2] = PR[GP1:90,2] + -9.859;
   1:L PR[91] R[100]mm/sec CNT100;
   1:  PR[GP1:91,1] = PR[GP1:90,1] + 50.670;
   1:  PR[GP1:91,2] = PR[GP1:90,2] + -0.085;
   1:L PR[91] R[100]mm/sec CNT100;
   1:  PR[GP1:91,1] = PR[GP1:90,1] + 49.915;
   1:  PR[GP1:91,2] = PR[GP1:90,2] + 4.045;
   1:L PR[91] R[100]mm/sec CNT100;
   1:  PR[GP1:91,1] = PR[GP1:90,1] + 48.539;
   1:  PR[GP1:91,2] = PR[GP1:90,2] + 13.913;
   1:L PR[91] R[100]mm/sec CNT100;
   1:  PR[GP1:91,1] = PR[GP1:90,1] + 44.535;
   1:  PR[GP1:91,2] = PR[GP1:90,2] + 22.982;
   1:L PR[91] R[100]mm/sec CNT100;
   1:  PR[GP1:91,1] = PR[GP1:90,1] + 42.388;
   1:  PR[GP1:91,2] = PR[GP1:90,2] + 26.568;
   1:L PR[91] R[100]mm/sec CNT100;
   1:  PR[GP1:91,1] = PR[GP1:90,1] + 35.981;
   1:  PR[GP1:91,2] = PR[GP1:90,2] + 34.286;
   1:L PR[91] R[100]mm/sec CNT100;
   1:  PR[GP1:91,1] = PR[GP1:90,1] + 32.830;
   1:  PR[GP1:91,2] = PR[GP1:90,2] + 36.814;
   1:L PR[91] R[100]mm/sec CNT100;
   1:  PR[GP1:91,1] = PR[GP1:90,1] + 25.435;
   1:  PR[GP1:91,2] = PR[GP1:90,2] + 42.051;
   1:L PR[91] R[100]mm/sec CNT100;
   1:  PR[GP1:91,1] = PR[GP1:90,1] + 16.981;
   1:  PR[GP1:91,2] = PR[GP1:90,2] + 45.327;
   1:L PR[91] R[100]mm/sec CNT100;
   1:  PR[GP1:91,1] = PR[GP1:90,1] + 13.219;
   1:  PR[GP1:91,2] = PR[GP1:90,2] + 46.593;
   1:L PR[91] R[100]mm/sec CNT100;
   1:  PR[GP1:91,1] = PR[GP1:90,1] + 4.090;
   1:  PR[GP1:91,2] = PR[GP1:90,2] + 47.723;
   1:L PR[91] R[100]mm/sec CNT100;
   1:  PR[GP1:91,1] = PR[GP1:90,1] + -0.114;
   1:  PR[GP1:91,2] = PR[GP1:90,2] + 47.642;
   1:L PR[91] R[100]mm/sec CNT100;
   1:  ! -- Layer/Ebene 200 -- !;
   1:  PR[91] = PR[90];
   1:  PR[GP1:91,1] = PR[GP1:90,1] + -3.510;
   1:  PR[GP1:91,2] = PR[GP1:90,2] + 47.871;
   1:  PR[GP1:91,3] = PR[GP1:90,3] + 122.305;
   1:L PR[91] R[100]mm/sec CNT100;
   1:  PR[GP1:91,1] = PR[GP1:90,1] + -12.910;
   1:  PR[GP1:91,2] = PR[GP1:90,2] + 46.707;
   1:L PR[91] R[100]mm/sec CNT100;
   1:  PR[GP1:91,1] = PR[GP1:90,1] + -16.319;
   1:  PR[GP1:91,2] = PR[GP1:90,2] + 45.559;
   1:L PR[91] R[100]mm/sec CNT100;
   1:  PR[GP1:91,1] = PR[GP1:90,1] + -25.024;
   1:  PR[GP1:91,2] = PR[GP1:90,2] + 42.186;
   1:L PR[91] R[100]mm/sec CNT100;
   1:  PR[GP1:91,1] = PR[GP1:90,1] + -27.980;
   1:  PR[GP1:91,2] = PR[GP1:90,2] + 39.825;
   1:L PR[91] R[100]mm/sec CNT100;
   1:  PR[GP1:91,1] = PR[GP1:90,1] + -35.537;
   1:  PR[GP1:91,2] = PR[GP1:90,2] + 34.473;
   1:L PR[91] R[100]mm/sec CNT100;
   1:  PR[GP1:91,1] = PR[GP1:90,1] + -42.150;
   1:  PR[GP1:91,2] = PR[GP1:90,2] + 26.508;
   1:L PR[91] R[100]mm/sec CNT100;
   1:  PR[GP1:91,1] = PR[GP1:90,1] + -44.096;
   1:  PR[GP1:91,2] = PR[GP1:90,2] + 23.258;
   1:L PR[91] R[100]mm/sec CNT100;
   1:  PR[GP1:91,1] = PR[GP1:90,1] + -48.245;
   1:  PR[GP1:91,2] = PR[GP1:90,2] + 13.857;
   1:L PR[91] R[100]mm/sec CNT100;
   1:  PR[GP1:91,1] = PR[GP1:90,1] + -48.937;
   1:  PR[GP1:91,2] = PR[GP1:90,2] + 10.066;
   1:L PR[91] R[100]mm/sec CNT100;
   1:  PR[GP1:91,1] = PR[GP1:90,1] + -50.349;
   1:  PR[GP1:91,2] = PR[GP1:90,2] + -0.059;
   1:L PR[91] R[100]mm/sec CNT100;
   1:  PR[GP1:91,1] = PR[GP1:90,1] + -49.665;
   1:  PR[GP1:91,2] = PR[GP1:90,2] + -3.798;
   1:L PR[91] R[100]mm/sec CNT100;
   1:  PR[GP1:91,1] = PR[GP1:90,1] + -48.240;
   1:  PR[GP1:91,2] = PR[GP1:90,2] + -14.013;
   1:L PR[91] R[100]mm/sec CNT100;
   1:  PR[GP1:91,1] = PR[GP1:90,1] + -44.096;
   1:  PR[GP1:91,2] = PR[GP1:90,2] + -23.401;
   1:L PR[91] R[100]mm/sec CNT100;
   1:  PR[GP1:91,1] = PR[GP1:90,1] + -42.150;
   1:  PR[GP1:91,2] = PR[GP1:90,2] + -26.652;
   1:L PR[91] R[100]mm/sec CNT100;
   1:  PR[GP1:91,1] = PR[GP1:90,1] + -35.526;
   1:  PR[GP1:91,2] = PR[GP1:90,2] + -34.631;
   1:L PR[91] R[100]mm/sec CNT100;
   1:  PR[GP1:91,1] = PR[GP1:90,1] + -32.672;
   1:  PR[GP1:91,2] = PR[GP1:90,2] + -36.920;
   1:L PR[91] R[100]mm/sec CNT100;
   1:  PR[GP1:91,1] = PR[GP1:90,1] + -25.042;
   1:  PR[GP1:91,2] = PR[GP1:90,2] + -42.323;
   1:L PR[91] R[100]mm/sec CNT100;
   1:  PR[GP1:91,1] = PR[GP1:90,1] + -16.320;
   1:  PR[GP1:91,2] = PR[GP1:90,2] + -45.703;
   1:L PR[91] R[100]mm/sec CNT100;
   1:  PR[GP1:91,1] = PR[GP1:90,1] + -12.911;
   1:  PR[GP1:91,2] = PR[GP1:90,2] + -46.850;
   1:L PR[91] R[100]mm/sec CNT100;
   1:  PR[GP1:91,1] = PR[GP1:90,1] + -3.511;
   1:  PR[GP1:91,2] = PR[GP1:90,2] + -48.015;
   1:L PR[91] R[100]mm/sec CNT100;
   1:  PR[GP1:91,1] = PR[GP1:90,1] + -0.094;
   1:  PR[GP1:91,2] = PR[GP1:90,2] + -47.942;
   1:L PR[91] R[100]mm/sec CNT100;
   1:  PR[GP1:91,1] = PR[GP1:90,1] + 3.721;
   1:  PR[GP1:91,2] = PR[GP1:90,2] + -48.015;
   1:L PR[91] R[100]mm/sec CNT100;
   1:  PR[GP1:91,1] = PR[GP1:90,1] + 13.123;
   1:  PR[GP1:91,2] = PR[GP1:90,2] + -46.851;
   1:L PR[91] R[100]mm/sec CNT100;
   1:  PR[GP1:91,1] = PR[GP1:90,1] + 16.532;
   1:  PR[GP1:91,2] = PR[GP1:90,2] + -45.703;
   1:L PR[91] R[100]mm/sec CNT100;
   1:  PR[GP1:91,1] = PR[GP1:90,1] + 25.238;
   1:  PR[GP1:91,2] = PR[GP1:90,2] + -42.329;
   1:L PR[91] R[100]mm/sec CNT100;
   1:  PR[GP1:91,1] = PR[GP1:90,1] + 28.193;
   1:  PR[GP1:91,2] = PR[GP1:90,2] + -39.968;
   1:L PR[91] R[100]mm/sec CNT100;
   1:  PR[GP1:91,1] = PR[GP1:90,1] + 35.752;
   1:  PR[GP1:91,2] = PR[GP1:90,2] + -34.615;
   1:L PR[91] R[100]mm/sec CNT100;
   1:  PR[GP1:91,1] = PR[GP1:90,1] + 42.364;
   1:  PR[GP1:91,2] = PR[GP1:90,2] + -26.650;
   1:L PR[91] R[100]mm/sec CNT100;
   1:  PR[GP1:91,1] = PR[GP1:90,1] + 44.309;
   1:  PR[GP1:91,2] = PR[GP1:90,2] + -23.402;
   1:L PR[91] R[100]mm/sec CNT100;
   1:  PR[GP1:91,1] = PR[GP1:90,1] + 48.459;
   1:  PR[GP1:91,2] = PR[GP1:90,2] + -14.002;
   1:L PR[91] R[100]mm/sec CNT100;
   1:  PR[GP1:91,1] = PR[GP1:90,1] + 49.150;
   1:  PR[GP1:91,2] = PR[GP1:90,2] + -10.209;
   1:L PR[91] R[100]mm/sec CNT100;
   1:  PR[GP1:91,1] = PR[GP1:90,1] + 50.562;
   1:  PR[GP1:91,2] = PR[GP1:90,2] + -0.085;
   1:L PR[91] R[100]mm/sec CNT100;
   1:  PR[GP1:91,1] = PR[GP1:90,1] + 49.878;
   1:  PR[GP1:91,2] = PR[GP1:90,2] + 3.656;
   1:L PR[91] R[100]mm/sec CNT100;
   1:  PR[GP1:91,1] = PR[GP1:90,1] + 48.454;
   1:  PR[GP1:91,2] = PR[GP1:90,2] + 13.870;
   1:L PR[91] R[100]mm/sec CNT100;
   1:  PR[GP1:91,1] = PR[GP1:90,1] + 44.309;
   1:  PR[GP1:91,2] = PR[GP1:90,2] + 23.258;
   1:L PR[91] R[100]mm/sec CNT100;
   1:  PR[GP1:91,1] = PR[GP1:90,1] + 42.364;
   1:  PR[GP1:91,2] = PR[GP1:90,2] + 26.507;
   1:L PR[91] R[100]mm/sec CNT100;
   1:  PR[GP1:91,1] = PR[GP1:90,1] + 35.741;
   1:  PR[GP1:91,2] = PR[GP1:90,2] + 34.485;
   1:L PR[91] R[100]mm/sec CNT100;
   1:  PR[GP1:91,1] = PR[GP1:90,1] + 32.886;
   1:  PR[GP1:91,2] = PR[GP1:90,2] + 36.776;
   1:L PR[91] R[100]mm/sec CNT100;
   1:  PR[GP1:91,1] = PR[GP1:90,1] + 25.254;
   1:  PR[GP1:91,2] = PR[GP1:90,2] + 42.179;
   1:L PR[91] R[100]mm/sec CNT100;
   1:  PR[GP1:91,1] = PR[GP1:90,1] + 16.531;
   1:  PR[GP1:91,2] = PR[GP1:90,2] + 45.560;
   1:L PR[91] R[100]mm/sec CNT100;
   1:  PR[GP1:91,1] = PR[GP1:90,1] + 13.122;
   1:  PR[GP1:91,2] = PR[GP1:90,2] + 46.707;
   1:L PR[91] R[100]mm/sec CNT100;
   1:  PR[GP1:91,1] = PR[GP1:90,1] + 3.720;
   1:  PR[GP1:91,2] = PR[GP1:90,2] + 47.871;
   1:L PR[91] R[100]mm/sec CNT100;
   1:  PR[GP1:91,1] = PR[GP1:90,1] + -0.094;
   1:  PR[GP1:91,2] = PR[GP1:90,2] + 47.798;
   1:L PR[91] R[100]mm/sec CNT100;
   1:  ! -- Layer/Ebene 201 -- !;
   1:  PR[91] = PR[90];
   1:  PR[GP1:91,1] = PR[GP1:90,1] + -3.139;
   1:  PR[GP1:91,2] = PR[GP1:90,2] + 48.019;
   1:  PR[GP1:91,3] = PR[GP1:90,3] + 122.915;
   1:L PR[91] R[100]mm/sec CNT100;
   1:  PR[GP1:91,1] = PR[GP1:90,1] + -12.814;
   1:  PR[GP1:91,2] = PR[GP1:90,2] + 46.821;
   1:L PR[91] R[100]mm/sec CNT100;
   1:  PR[GP1:91,1] = PR[GP1:90,1] + -15.869;
   1:  PR[GP1:91,2] = PR[GP1:90,2] + 45.792;
   1:L PR[91] R[100]mm/sec CNT100;
   1:  PR[GP1:91,1] = PR[GP1:90,1] + -24.844;
   1:  PR[GP1:91,2] = PR[GP1:90,2] + 42.314;
   1:L PR[91] R[100]mm/sec CNT100;
   1:  PR[GP1:91,1] = PR[GP1:90,1] + -27.493;
   1:  PR[GP1:91,2] = PR[GP1:90,2] + 40.198;
   1:L PR[91] R[100]mm/sec CNT100;
   1:  PR[GP1:91,1] = PR[GP1:90,1] + -35.297;
   1:  PR[GP1:91,2] = PR[GP1:90,2] + 34.672;
   1:L PR[91] R[100]mm/sec CNT100;
   1:  PR[GP1:91,1] = PR[GP1:90,1] + -42.126;
   1:  PR[GP1:91,2] = PR[GP1:90,2] + 26.446;
   1:L PR[91] R[100]mm/sec CNT100;
   1:  PR[GP1:91,1] = PR[GP1:90,1] + -43.870;
   1:  PR[GP1:91,2] = PR[GP1:90,2] + 23.533;
   1:L PR[91] R[100]mm/sec CNT100;
   1:  PR[GP1:91,1] = PR[GP1:90,1] + -48.160;
   1:  PR[GP1:91,2] = PR[GP1:90,2] + 13.814;
   1:L PR[91] R[100]mm/sec CNT100;
   1:  PR[GP1:91,1] = PR[GP1:90,1] + -48.780;
   1:  PR[GP1:91,2] = PR[GP1:90,2] + 10.416;
   1:L PR[91] R[100]mm/sec CNT100;
   1:  PR[GP1:91,1] = PR[GP1:90,1] + -50.241;
   1:  PR[GP1:91,2] = PR[GP1:90,2] + -0.059;
   1:L PR[91] R[100]mm/sec CNT100;
   1:  PR[GP1:91,1] = PR[GP1:90,1] + -49.628;
   1:  PR[GP1:91,2] = PR[GP1:90,2] + -3.410;
   1:L PR[91] R[100]mm/sec CNT100;
   1:  PR[GP1:91,1] = PR[GP1:90,1] + -48.155;
   1:  PR[GP1:91,2] = PR[GP1:90,2] + -13.970;
   1:L PR[91] R[100]mm/sec CNT100;
   1:  PR[GP1:91,1] = PR[GP1:90,1] + -43.870;
   1:  PR[GP1:91,2] = PR[GP1:90,2] + -23.677;
   1:L PR[91] R[100]mm/sec CNT100;
   1:  PR[GP1:91,1] = PR[GP1:90,1] + -42.126;
   1:  PR[GP1:91,2] = PR[GP1:90,2] + -26.590;
   1:L PR[91] R[100]mm/sec CNT100;
   1:  PR[GP1:91,1] = PR[GP1:90,1] + -35.285;
   1:  PR[GP1:91,2] = PR[GP1:90,2] + -34.830;
   1:L PR[91] R[100]mm/sec CNT100;
   1:  PR[GP1:91,1] = PR[GP1:90,1] + -32.728;
   1:  PR[GP1:91,2] = PR[GP1:90,2] + -36.881;
   1:L PR[91] R[100]mm/sec CNT100;
   1:  PR[GP1:91,1] = PR[GP1:90,1] + -24.861;
   1:  PR[GP1:91,2] = PR[GP1:90,2] + -42.452;
   1:L PR[91] R[100]mm/sec CNT100;
   1:  PR[GP1:91,1] = PR[GP1:90,1] + -15.869;
   1:  PR[GP1:91,2] = PR[GP1:90,2] + -45.936;
   1:L PR[91] R[100]mm/sec CNT100;
   1:  PR[GP1:91,1] = PR[GP1:90,1] + -12.814;
   1:  PR[GP1:91,2] = PR[GP1:90,2] + -46.965;
   1:L PR[91] R[100]mm/sec CNT100;
   1:  PR[GP1:91,1] = PR[GP1:90,1] + -3.140;
   1:  PR[GP1:91,2] = PR[GP1:90,2] + -48.163;
   1:L PR[91] R[100]mm/sec CNT100;
   1:  PR[GP1:91,1] = PR[GP1:90,1] + -0.074;
   1:  PR[GP1:91,2] = PR[GP1:90,2] + -48.097;
   1:L PR[91] R[100]mm/sec CNT100;
   1:  PR[GP1:91,1] = PR[GP1:90,1] + 3.350;
   1:  PR[GP1:91,2] = PR[GP1:90,2] + -48.163;
   1:L PR[91] R[100]mm/sec CNT100;
   1:  PR[GP1:91,1] = PR[GP1:90,1] + 13.026;
   1:  PR[GP1:91,2] = PR[GP1:90,2] + -46.965;
   1:L PR[91] R[100]mm/sec CNT100;
   1:  PR[GP1:91,1] = PR[GP1:90,1] + 16.081;
   1:  PR[GP1:91,2] = PR[GP1:90,2] + -45.936;
   1:L PR[91] R[100]mm/sec CNT100;
   1:  PR[GP1:91,1] = PR[GP1:90,1] + 25.058;
   1:  PR[GP1:91,2] = PR[GP1:90,2] + -42.458;
   1:L PR[91] R[100]mm/sec CNT100;
   1:  PR[GP1:91,1] = PR[GP1:90,1] + 27.706;
   1:  PR[GP1:91,2] = PR[GP1:90,2] + -40.341;
   1:L PR[91] R[100]mm/sec CNT100;
   1:  PR[GP1:91,1] = PR[GP1:90,1] + 35.512;
   1:  PR[GP1:91,2] = PR[GP1:90,2] + -34.814;
   1:L PR[91] R[100]mm/sec CNT100;
   1:  PR[GP1:91,1] = PR[GP1:90,1] + 42.340;
   1:  PR[GP1:91,2] = PR[GP1:90,2] + -26.588;
   1:L PR[91] R[100]mm/sec CNT100;
   1:  PR[GP1:91,1] = PR[GP1:90,1] + 44.083;
   1:  PR[GP1:91,2] = PR[GP1:90,2] + -23.677;
   1:L PR[91] R[100]mm/sec CNT100;
   1:  PR[GP1:91,1] = PR[GP1:90,1] + 48.374;
   1:  PR[GP1:91,2] = PR[GP1:90,2] + -13.959;
   1:L PR[91] R[100]mm/sec CNT100;
   1:  PR[GP1:91,1] = PR[GP1:90,1] + 48.993;
   1:  PR[GP1:91,2] = PR[GP1:90,2] + -10.560;
   1:L PR[91] R[100]mm/sec CNT100;
   1:  PR[GP1:91,1] = PR[GP1:90,1] + 50.454;
   1:  PR[GP1:91,2] = PR[GP1:90,2] + -0.085;
   1:L PR[91] R[100]mm/sec CNT100;
   1:  PR[GP1:91,1] = PR[GP1:90,1] + 49.841;
   1:  PR[GP1:91,2] = PR[GP1:90,2] + 3.267;
   1:L PR[91] R[100]mm/sec CNT100;
   1:  PR[GP1:91,1] = PR[GP1:90,1] + 48.369;
   1:  PR[GP1:91,2] = PR[GP1:90,2] + 13.827;
   1:L PR[91] R[100]mm/sec CNT100;
   1:  PR[GP1:91,1] = PR[GP1:90,1] + 44.083;
   1:  PR[GP1:91,2] = PR[GP1:90,2] + 23.533;
   1:L PR[91] R[100]mm/sec CNT100;
   1:  PR[GP1:91,1] = PR[GP1:90,1] + 42.340;
   1:  PR[GP1:91,2] = PR[GP1:90,2] + 26.445;
   1:L PR[91] R[100]mm/sec CNT100;
   1:  PR[GP1:91,1] = PR[GP1:90,1] + 35.500;
   1:  PR[GP1:91,2] = PR[GP1:90,2] + 34.684;
   1:L PR[91] R[100]mm/sec CNT100;
   1:  PR[GP1:91,1] = PR[GP1:90,1] + 32.942;
   1:  PR[GP1:91,2] = PR[GP1:90,2] + 36.737;
   1:L PR[91] R[100]mm/sec CNT100;
   1:  PR[GP1:91,1] = PR[GP1:90,1] + 25.074;
   1:  PR[GP1:91,2] = PR[GP1:90,2] + 42.308;
   1:L PR[91] R[100]mm/sec CNT100;
   1:  PR[GP1:91,1] = PR[GP1:90,1] + 16.081;
   1:  PR[GP1:91,2] = PR[GP1:90,2] + 45.793;
   1:L PR[91] R[100]mm/sec CNT100;
   1:  PR[GP1:91,1] = PR[GP1:90,1] + 13.026;
   1:  PR[GP1:91,2] = PR[GP1:90,2] + 46.821;
   1:L PR[91] R[100]mm/sec CNT100;
   1:  PR[GP1:91,1] = PR[GP1:90,1] + 3.349;
   1:  PR[GP1:91,2] = PR[GP1:90,2] + 48.019;
   1:L PR[91] R[100]mm/sec CNT100;
   1:  PR[GP1:91,1] = PR[GP1:90,1] + -0.074;
   1:  PR[GP1:91,2] = PR[GP1:90,2] + 47.953;
   1:L PR[91] R[100]mm/sec CNT100;
   1:  ! -- Layer/Ebene 202 -- !;
   1:  PR[91] = PR[90];
   1:  PR[GP1:91,1] = PR[GP1:90,1] + -2.769;
   1:  PR[GP1:91,2] = PR[GP1:90,2] + 48.167;
   1:  PR[GP1:91,3] = PR[GP1:90,3] + 123.525;
   1:L PR[91] R[100]mm/sec CNT100;
   1:  PR[GP1:91,1] = PR[GP1:90,1] + -12.717;
   1:  PR[GP1:91,2] = PR[GP1:90,2] + 46.935;
   1:L PR[91] R[100]mm/sec CNT100;
   1:  PR[GP1:91,1] = PR[GP1:90,1] + -15.418;
   1:  PR[GP1:91,2] = PR[GP1:90,2] + 46.026;
   1:L PR[91] R[100]mm/sec CNT100;
   1:  PR[GP1:91,1] = PR[GP1:90,1] + -24.664;
   1:  PR[GP1:91,2] = PR[GP1:90,2] + 42.443;
   1:L PR[91] R[100]mm/sec CNT100;
   1:  PR[GP1:91,1] = PR[GP1:90,1] + -27.006;
   1:  PR[GP1:91,2] = PR[GP1:90,2] + 40.571;
   1:L PR[91] R[100]mm/sec CNT100;
   1:  PR[GP1:91,1] = PR[GP1:90,1] + -35.056;
   1:  PR[GP1:91,2] = PR[GP1:90,2] + 34.871;
   1:L PR[91] R[100]mm/sec CNT100;
   1:  PR[GP1:91,1] = PR[GP1:90,1] + -42.102;
   1:  PR[GP1:91,2] = PR[GP1:90,2] + 26.384;
   1:L PR[91] R[100]mm/sec CNT100;
   1:  PR[GP1:91,1] = PR[GP1:90,1] + -43.644;
   1:  PR[GP1:91,2] = PR[GP1:90,2] + 23.809;
   1:L PR[91] R[100]mm/sec CNT100;
   1:  PR[GP1:91,1] = PR[GP1:90,1] + -48.075;
   1:  PR[GP1:91,2] = PR[GP1:90,2] + 13.771;
   1:L PR[91] R[100]mm/sec CNT100;
   1:  PR[GP1:91,1] = PR[GP1:90,1] + -48.623;
   1:  PR[GP1:91,2] = PR[GP1:90,2] + 10.767;
   1:L PR[91] R[100]mm/sec CNT100;
   1:  PR[GP1:91,1] = PR[GP1:90,1] + -50.133;
   1:  PR[GP1:91,2] = PR[GP1:90,2] + -0.059;
   1:L PR[91] R[100]mm/sec CNT100;
   1:  PR[GP1:91,1] = PR[GP1:90,1] + -49.591;
   1:  PR[GP1:91,2] = PR[GP1:90,2] + -3.021;
   1:L PR[91] R[100]mm/sec CNT100;
   1:  PR[GP1:91,1] = PR[GP1:90,1] + -48.070;
   1:  PR[GP1:91,2] = PR[GP1:90,2] + -13.926;
   1:L PR[91] R[100]mm/sec CNT100;
   1:  PR[GP1:91,1] = PR[GP1:90,1] + -43.644;
   1:  PR[GP1:91,2] = PR[GP1:90,2] + -23.953;
   1:L PR[91] R[100]mm/sec CNT100;
   1:  PR[GP1:91,1] = PR[GP1:90,1] + -42.102;
   1:  PR[GP1:91,2] = PR[GP1:90,2] + -26.528;
   1:L PR[91] R[100]mm/sec CNT100;
   1:  PR[GP1:91,1] = PR[GP1:90,1] + -35.045;
   1:  PR[GP1:91,2] = PR[GP1:90,2] + -35.029;
   1:L PR[91] R[100]mm/sec CNT100;
   1:  PR[GP1:91,1] = PR[GP1:90,1] + -32.784;
   1:  PR[GP1:91,2] = PR[GP1:90,2] + -36.842;
   1:L PR[91] R[100]mm/sec CNT100;
   1:  PR[GP1:91,1] = PR[GP1:90,1] + -24.681;
   1:  PR[GP1:91,2] = PR[GP1:90,2] + -42.580;
   1:L PR[91] R[100]mm/sec CNT100;
   1:  PR[GP1:91,1] = PR[GP1:90,1] + -15.419;
   1:  PR[GP1:91,2] = PR[GP1:90,2] + -46.169;
   1:L PR[91] R[100]mm/sec CNT100;
   1:  PR[GP1:91,1] = PR[GP1:90,1] + -12.718;
   1:  PR[GP1:91,2] = PR[GP1:90,2] + -47.079;
   1:L PR[91] R[100]mm/sec CNT100;
   1:  PR[GP1:91,1] = PR[GP1:90,1] + -2.769;
   1:  PR[GP1:91,2] = PR[GP1:90,2] + -48.311;
   1:L PR[91] R[100]mm/sec CNT100;
   1:  PR[GP1:91,1] = PR[GP1:90,1] + -0.054;
   1:  PR[GP1:91,2] = PR[GP1:90,2] + -48.253;
   1:L PR[91] R[100]mm/sec CNT100;
   1:  PR[GP1:91,1] = PR[GP1:90,1] + 2.979;
   1:  PR[GP1:91,2] = PR[GP1:90,2] + -48.311;
   1:L PR[91] R[100]mm/sec CNT100;
   1:  PR[GP1:91,1] = PR[GP1:90,1] + 12.930;
   1:  PR[GP1:91,2] = PR[GP1:90,2] + -47.079;
   1:L PR[91] R[100]mm/sec CNT100;
   1:  PR[GP1:91,1] = PR[GP1:90,1] + 15.631;
   1:  PR[GP1:91,2] = PR[GP1:90,2] + -46.170;
   1:L PR[91] R[100]mm/sec CNT100;
   1:  PR[GP1:91,1] = PR[GP1:90,1] + 24.878;
   1:  PR[GP1:91,2] = PR[GP1:90,2] + -42.587;
   1:L PR[91] R[100]mm/sec CNT100;
   1:  PR[GP1:91,1] = PR[GP1:90,1] + 27.220;
   1:  PR[GP1:91,2] = PR[GP1:90,2] + -40.714;
   1:L PR[91] R[100]mm/sec CNT100;
   1:  PR[GP1:91,1] = PR[GP1:90,1] + 35.272;
   1:  PR[GP1:91,2] = PR[GP1:90,2] + -35.013;
   1:L PR[91] R[100]mm/sec CNT100;
   1:  PR[GP1:91,1] = PR[GP1:90,1] + 42.316;
   1:  PR[GP1:91,2] = PR[GP1:90,2] + -26.526;
   1:L PR[91] R[100]mm/sec CNT100;
   1:  PR[GP1:91,1] = PR[GP1:90,1] + 43.857;
   1:  PR[GP1:91,2] = PR[GP1:90,2] + -23.953;
   1:L PR[91] R[100]mm/sec CNT100;
   1:  PR[GP1:91,1] = PR[GP1:90,1] + 48.289;
   1:  PR[GP1:91,2] = PR[GP1:90,2] + -13.915;
   1:L PR[91] R[100]mm/sec CNT100;
   1:  PR[GP1:91,1] = PR[GP1:90,1] + 48.836;
   1:  PR[GP1:91,2] = PR[GP1:90,2] + -10.910;
   1:L PR[91] R[100]mm/sec CNT100;
   1:  PR[GP1:91,1] = PR[GP1:90,1] + 50.346;
   1:  PR[GP1:91,2] = PR[GP1:90,2] + -0.085;
   1:L PR[91] R[100]mm/sec CNT100;
   1:  PR[GP1:91,1] = PR[GP1:90,1] + 49.804;
   1:  PR[GP1:91,2] = PR[GP1:90,2] + 2.879;
   1:L PR[91] R[100]mm/sec CNT100;
   1:  PR[GP1:91,1] = PR[GP1:90,1] + 48.283;
   1:  PR[GP1:91,2] = PR[GP1:90,2] + 13.783;
   1:L PR[91] R[100]mm/sec CNT100;
   1:  PR[GP1:91,1] = PR[GP1:90,1] + 43.857;
   1:  PR[GP1:91,2] = PR[GP1:90,2] + 23.809;
   1:L PR[91] R[100]mm/sec CNT100;
   1:  PR[GP1:91,1] = PR[GP1:90,1] + 42.316;
   1:  PR[GP1:91,2] = PR[GP1:90,2] + 26.383;
   1:L PR[91] R[100]mm/sec CNT100;
   1:  PR[GP1:91,1] = PR[GP1:90,1] + 35.260;
   1:  PR[GP1:91,2] = PR[GP1:90,2] + 34.883;
   1:L PR[91] R[100]mm/sec CNT100;
   1:  PR[GP1:91,1] = PR[GP1:90,1] + 32.998;
   1:  PR[GP1:91,2] = PR[GP1:90,2] + 36.698;
   1:L PR[91] R[100]mm/sec CNT100;
   1:  PR[GP1:91,1] = PR[GP1:90,1] + 24.894;
   1:  PR[GP1:91,2] = PR[GP1:90,2] + 42.436;
   1:L PR[91] R[100]mm/sec CNT100;
   1:  PR[GP1:91,1] = PR[GP1:90,1] + 15.630;
   1:  PR[GP1:91,2] = PR[GP1:90,2] + 46.026;
   1:L PR[91] R[100]mm/sec CNT100;
   1:  PR[GP1:91,1] = PR[GP1:90,1] + 12.929;
   1:  PR[GP1:91,2] = PR[GP1:90,2] + 46.935;
   1:L PR[91] R[100]mm/sec CNT100;
   1:  PR[GP1:91,1] = PR[GP1:90,1] + 2.978;
   1:  PR[GP1:91,2] = PR[GP1:90,2] + 48.167;
   1:L PR[91] R[100]mm/sec CNT100;
   1:  PR[GP1:91,1] = PR[GP1:90,1] + -0.054;
   1:  PR[GP1:91,2] = PR[GP1:90,2] + 48.109;
   1:L PR[91] R[100]mm/sec CNT100;
   1:  ! -- Layer/Ebene 203 -- !;
   1:  PR[91] = PR[90];
   1:  PR[GP1:91,1] = PR[GP1:90,1] + -2.398;
   1:  PR[GP1:91,2] = PR[GP1:90,2] + 48.315;
   1:  PR[GP1:91,3] = PR[GP1:90,3] + 124.135;
   1:L PR[91] R[100]mm/sec CNT100;
   1:  PR[GP1:91,1] = PR[GP1:90,1] + -12.620;
   1:  PR[GP1:91,2] = PR[GP1:90,2] + 47.049;
   1:L PR[91] R[100]mm/sec CNT100;
   1:  PR[GP1:91,1] = PR[GP1:90,1] + -14.968;
   1:  PR[GP1:91,2] = PR[GP1:90,2] + 46.259;
   1:L PR[91] R[100]mm/sec CNT100;
   1:  PR[GP1:91,1] = PR[GP1:90,1] + -24.484;
   1:  PR[GP1:91,2] = PR[GP1:90,2] + 42.571;
   1:L PR[91] R[100]mm/sec CNT100;
   1:  PR[GP1:91,1] = PR[GP1:90,1] + -26.520;
   1:  PR[GP1:91,2] = PR[GP1:90,2] + 40.944;
   1:L PR[91] R[100]mm/sec CNT100;
   1:  PR[GP1:91,1] = PR[GP1:90,1] + -34.816;
   1:  PR[GP1:91,2] = PR[GP1:90,2] + 35.070;
   1:L PR[91] R[100]mm/sec CNT100;
   1:  PR[GP1:91,1] = PR[GP1:90,1] + -42.078;
   1:  PR[GP1:91,2] = PR[GP1:90,2] + 26.322;
   1:L PR[91] R[100]mm/sec CNT100;
   1:  PR[GP1:91,1] = PR[GP1:90,1] + -43.418;
   1:  PR[GP1:91,2] = PR[GP1:90,2] + 24.085;
   1:L PR[91] R[100]mm/sec CNT100;
   1:  PR[GP1:91,1] = PR[GP1:90,1] + -47.990;
   1:  PR[GP1:91,2] = PR[GP1:90,2] + 13.728;
   1:L PR[91] R[100]mm/sec CNT100;
   1:  PR[GP1:91,1] = PR[GP1:90,1] + -48.466;
   1:  PR[GP1:91,2] = PR[GP1:90,2] + 11.117;
   1:L PR[91] R[100]mm/sec CNT100;
   1:  PR[GP1:91,1] = PR[GP1:90,1] + -50.025;
   1:  PR[GP1:91,2] = PR[GP1:90,2] + -0.059;
   1:L PR[91] R[100]mm/sec CNT100;
   1:  PR[GP1:91,1] = PR[GP1:90,1] + -49.554;
   1:  PR[GP1:91,2] = PR[GP1:90,2] + -2.633;
   1:L PR[91] R[100]mm/sec CNT100;
   1:  PR[GP1:91,1] = PR[GP1:90,1] + -47.985;
   1:  PR[GP1:91,2] = PR[GP1:90,2] + -13.883;
   1:L PR[91] R[100]mm/sec CNT100;
   1:  PR[GP1:91,1] = PR[GP1:90,1] + -43.418;
   1:  PR[GP1:91,2] = PR[GP1:90,2] + -24.229;
   1:L PR[91] R[100]mm/sec CNT100;
   1:  PR[GP1:91,1] = PR[GP1:90,1] + -42.079;
   1:  PR[GP1:91,2] = PR[GP1:90,2] + -26.466;
   1:L PR[91] R[100]mm/sec CNT100;
   1:  PR[GP1:91,1] = PR[GP1:90,1] + -34.804;
   1:  PR[GP1:91,2] = PR[GP1:90,2] + -35.228;
   1:L PR[91] R[100]mm/sec CNT100;
   1:  PR[GP1:91,1] = PR[GP1:90,1] + -32.840;
   1:  PR[GP1:91,2] = PR[GP1:90,2] + -36.803;
   1:L PR[91] R[100]mm/sec CNT100;
   1:  PR[GP1:91,1] = PR[GP1:90,1] + -24.500;
   1:  PR[GP1:91,2] = PR[GP1:90,2] + -42.709;
   1:L PR[91] R[100]mm/sec CNT100;
   1:  PR[GP1:91,1] = PR[GP1:90,1] + -14.969;
   1:  PR[GP1:91,2] = PR[GP1:90,2] + -46.402;
   1:L PR[91] R[100]mm/sec CNT100;
   1:  PR[GP1:91,1] = PR[GP1:90,1] + -12.621;
   1:  PR[GP1:91,2] = PR[GP1:90,2] + -47.193;
   1:L PR[91] R[100]mm/sec CNT100;
   1:  PR[GP1:91,1] = PR[GP1:90,1] + -2.399;
   1:  PR[GP1:91,2] = PR[GP1:90,2] + -48.459;
   1:L PR[91] R[100]mm/sec CNT100;
   1:  PR[GP1:91,1] = PR[GP1:90,1] + -0.034;
   1:  PR[GP1:91,2] = PR[GP1:90,2] + -48.408;
   1:L PR[91] R[100]mm/sec CNT100;
   1:  PR[GP1:91,1] = PR[GP1:90,1] + 2.608;
   1:  PR[GP1:91,2] = PR[GP1:90,2] + -48.459;
   1:L PR[91] R[100]mm/sec CNT100;
   1:  PR[GP1:91,1] = PR[GP1:90,1] + 12.833;
   1:  PR[GP1:91,2] = PR[GP1:90,2] + -47.193;
   1:L PR[91] R[100]mm/sec CNT100;
   1:  PR[GP1:91,1] = PR[GP1:90,1] + 15.180;
   1:  PR[GP1:91,2] = PR[GP1:90,2] + -46.403;
   1:L PR[91] R[100]mm/sec CNT100;
   1:  PR[GP1:91,1] = PR[GP1:90,1] + 24.697;
   1:  PR[GP1:91,2] = PR[GP1:90,2] + -42.715;
   1:L PR[91] R[100]mm/sec CNT100;
   1:  PR[GP1:91,1] = PR[GP1:90,1] + 26.733;
   1:  PR[GP1:91,2] = PR[GP1:90,2] + -41.088;
   1:L PR[91] R[100]mm/sec CNT100;
   1:  PR[GP1:91,1] = PR[GP1:90,1] + 35.031;
   1:  PR[GP1:91,2] = PR[GP1:90,2] + -35.212;
   1:L PR[91] R[100]mm/sec CNT100;
   1:  PR[GP1:91,1] = PR[GP1:90,1] + 42.292;
   1:  PR[GP1:91,2] = PR[GP1:90,2] + -26.464;
   1:L PR[91] R[100]mm/sec CNT100;
   1:  PR[GP1:91,1] = PR[GP1:90,1] + 43.631;
   1:  PR[GP1:91,2] = PR[GP1:90,2] + -24.228;
   1:L PR[91] R[100]mm/sec CNT100;
   1:  PR[GP1:91,1] = PR[GP1:90,1] + 48.203;
   1:  PR[GP1:91,2] = PR[GP1:90,2] + -13.872;
   1:L PR[91] R[100]mm/sec CNT100;
   1:  PR[GP1:91,1] = PR[GP1:90,1] + 48.679;
   1:  PR[GP1:91,2] = PR[GP1:90,2] + -11.261;
   1:L PR[91] R[100]mm/sec CNT100;
   1:  PR[GP1:91,1] = PR[GP1:90,1] + 50.238;
   1:  PR[GP1:91,2] = PR[GP1:90,2] + -0.085;
   1:L PR[91] R[100]mm/sec CNT100;
   1:  PR[GP1:91,1] = PR[GP1:90,1] + 49.767;
   1:  PR[GP1:91,2] = PR[GP1:90,2] + 2.490;
   1:L PR[91] R[100]mm/sec CNT100;
   1:  PR[GP1:91,1] = PR[GP1:90,1] + 48.198;
   1:  PR[GP1:91,2] = PR[GP1:90,2] + 13.740;
   1:L PR[91] R[100]mm/sec CNT100;
   1:  PR[GP1:91,1] = PR[GP1:90,1] + 43.631;
   1:  PR[GP1:91,2] = PR[GP1:90,2] + 24.085;
   1:L PR[91] R[100]mm/sec CNT100;
   1:  PR[GP1:91,1] = PR[GP1:90,1] + 42.292;
   1:  PR[GP1:91,2] = PR[GP1:90,2] + 26.321;
   1:L PR[91] R[100]mm/sec CNT100;
   1:  PR[GP1:91,1] = PR[GP1:90,1] + 35.019;
   1:  PR[GP1:91,2] = PR[GP1:90,2] + 35.082;
   1:L PR[91] R[100]mm/sec CNT100;
   1:  PR[GP1:91,1] = PR[GP1:90,1] + 33.054;
   1:  PR[GP1:91,2] = PR[GP1:90,2] + 36.659;
   1:L PR[91] R[100]mm/sec CNT100;
   1:  PR[GP1:91,1] = PR[GP1:90,1] + 24.713;
   1:  PR[GP1:91,2] = PR[GP1:90,2] + 42.565;
   1:L PR[91] R[100]mm/sec CNT100;
   1:  PR[GP1:91,1] = PR[GP1:90,1] + 15.180;
   1:  PR[GP1:91,2] = PR[GP1:90,2] + 46.259;
   1:L PR[91] R[100]mm/sec CNT100;
   1:  PR[GP1:91,1] = PR[GP1:90,1] + 12.832;
   1:  PR[GP1:91,2] = PR[GP1:90,2] + 47.049;
   1:L PR[91] R[100]mm/sec CNT100;
   1:  PR[GP1:91,1] = PR[GP1:90,1] + 2.608;
   1:  PR[GP1:91,2] = PR[GP1:90,2] + 48.315;
   1:L PR[91] R[100]mm/sec CNT100;
   1:  PR[GP1:91,1] = PR[GP1:90,1] + -0.034;
   1:  PR[GP1:91,2] = PR[GP1:90,2] + 48.264;
   1:L PR[91] R[100]mm/sec CNT100;
   1:  ! -- Layer/Ebene 204 -- !;
   1:  PR[91] = PR[90];
   1:  PR[GP1:91,1] = PR[GP1:90,1] + -2.027;
   1:  PR[GP1:91,2] = PR[GP1:90,2] + 48.463;
   1:  PR[GP1:91,3] = PR[GP1:90,3] + 124.745;
   1:L PR[91] R[100]mm/sec CNT100;
   1:  PR[GP1:91,1] = PR[GP1:90,1] + -12.524;
   1:  PR[GP1:91,2] = PR[GP1:90,2] + 47.163;
   1:L PR[91] R[100]mm/sec CNT100;
   1:  PR[GP1:91,1] = PR[GP1:90,1] + -14.518;
   1:  PR[GP1:91,2] = PR[GP1:90,2] + 46.492;
   1:L PR[91] R[100]mm/sec CNT100;
   1:  PR[GP1:91,1] = PR[GP1:90,1] + -24.303;
   1:  PR[GP1:91,2] = PR[GP1:90,2] + 42.700;
   1:L PR[91] R[100]mm/sec CNT100;
   1:  PR[GP1:91,1] = PR[GP1:90,1] + -26.033;
   1:  PR[GP1:91,2] = PR[GP1:90,2] + 41.318;
   1:L PR[91] R[100]mm/sec CNT100;
   1:  PR[GP1:91,1] = PR[GP1:90,1] + -34.575;
   1:  PR[GP1:91,2] = PR[GP1:90,2] + 35.269;
   1:L PR[91] R[100]mm/sec CNT100;
   1:  PR[GP1:91,1] = PR[GP1:90,1] + -42.055;
   1:  PR[GP1:91,2] = PR[GP1:90,2] + 26.260;
   1:L PR[91] R[100]mm/sec CNT100;
   1:  PR[GP1:91,1] = PR[GP1:90,1] + -43.192;
   1:  PR[GP1:91,2] = PR[GP1:90,2] + 24.360;
   1:L PR[91] R[100]mm/sec CNT100;
   1:  PR[GP1:91,1] = PR[GP1:90,1] + -47.905;
   1:  PR[GP1:91,2] = PR[GP1:90,2] + 13.685;
   1:L PR[91] R[100]mm/sec CNT100;
   1:  PR[GP1:91,1] = PR[GP1:90,1] + -48.309;
   1:  PR[GP1:91,2] = PR[GP1:90,2] + 11.468;
   1:L PR[91] R[100]mm/sec CNT100;
   1:  PR[GP1:91,1] = PR[GP1:90,1] + -49.917;
   1:  PR[GP1:91,2] = PR[GP1:90,2] + -0.059;
   1:L PR[91] R[100]mm/sec CNT100;
   1:  PR[GP1:91,1] = PR[GP1:90,1] + -49.517;
   1:  PR[GP1:91,2] = PR[GP1:90,2] + -2.244;
   1:L PR[91] R[100]mm/sec CNT100;
   1:  PR[GP1:91,1] = PR[GP1:90,1] + -47.900;
   1:  PR[GP1:91,2] = PR[GP1:90,2] + -13.840;
   1:L PR[91] R[100]mm/sec CNT100;
   1:  PR[GP1:91,1] = PR[GP1:90,1] + -43.192;
   1:  PR[GP1:91,2] = PR[GP1:90,2] + -24.504;
   1:L PR[91] R[100]mm/sec CNT100;
   1:  PR[GP1:91,1] = PR[GP1:90,1] + -42.055;
   1:  PR[GP1:91,2] = PR[GP1:90,2] + -26.404;
   1:L PR[91] R[100]mm/sec CNT100;
   1:  PR[GP1:91,1] = PR[GP1:90,1] + -34.564;
   1:  PR[GP1:91,2] = PR[GP1:90,2] + -35.426;
   1:L PR[91] R[100]mm/sec CNT100;
   1:  PR[GP1:91,1] = PR[GP1:90,1] + -32.896;
   1:  PR[GP1:91,2] = PR[GP1:90,2] + -36.764;
   1:L PR[91] R[100]mm/sec CNT100;
   1:  PR[GP1:91,1] = PR[GP1:90,1] + -24.320;
   1:  PR[GP1:91,2] = PR[GP1:90,2] + -42.837;
   1:L PR[91] R[100]mm/sec CNT100;
   1:  PR[GP1:91,1] = PR[GP1:90,1] + -14.518;
   1:  PR[GP1:91,2] = PR[GP1:90,2] + -46.636;
   1:L PR[91] R[100]mm/sec CNT100;
   1:  PR[GP1:91,1] = PR[GP1:90,1] + -12.524;
   1:  PR[GP1:91,2] = PR[GP1:90,2] + -47.307;
   1:L PR[91] R[100]mm/sec CNT100;
   1:  PR[GP1:91,1] = PR[GP1:90,1] + -2.028;
   1:  PR[GP1:91,2] = PR[GP1:90,2] + -48.607;
   1:L PR[91] R[100]mm/sec CNT100;
   1:  PR[GP1:91,1] = PR[GP1:90,1] + -0.014;
   1:  PR[GP1:91,2] = PR[GP1:90,2] + -48.564;
   1:L PR[91] R[100]mm/sec CNT100;
   1:  PR[GP1:91,1] = PR[GP1:90,1] + 2.237;
   1:  PR[GP1:91,2] = PR[GP1:90,2] + -48.607;
   1:L PR[91] R[100]mm/sec CNT100;
   1:  PR[GP1:91,1] = PR[GP1:90,1] + 12.736;
   1:  PR[GP1:91,2] = PR[GP1:90,2] + -47.307;
   1:L PR[91] R[100]mm/sec CNT100;
   1:  PR[GP1:91,1] = PR[GP1:90,1] + 14.730;
   1:  PR[GP1:91,2] = PR[GP1:90,2] + -46.636;
   1:L PR[91] R[100]mm/sec CNT100;
   1:  PR[GP1:91,1] = PR[GP1:90,1] + 24.517;
   1:  PR[GP1:91,2] = PR[GP1:90,2] + -42.844;
   1:L PR[91] R[100]mm/sec CNT100;
   1:  PR[GP1:91,1] = PR[GP1:90,1] + 26.246;
   1:  PR[GP1:91,2] = PR[GP1:90,2] + -41.461;
   1:L PR[91] R[100]mm/sec CNT100;
   1:  PR[GP1:91,1] = PR[GP1:90,1] + 34.791;
   1:  PR[GP1:91,2] = PR[GP1:90,2] + -35.411;
   1:L PR[91] R[100]mm/sec CNT100;
   1:  PR[GP1:91,1] = PR[GP1:90,1] + 42.269;
   1:  PR[GP1:91,2] = PR[GP1:90,2] + -26.403;
   1:L PR[91] R[100]mm/sec CNT100;
   1:  PR[GP1:91,1] = PR[GP1:90,1] + 43.405;
   1:  PR[GP1:91,2] = PR[GP1:90,2] + -24.504;
   1:L PR[91] R[100]mm/sec CNT100;
   1:  PR[GP1:91,1] = PR[GP1:90,1] + 48.118;
   1:  PR[GP1:91,2] = PR[GP1:90,2] + -13.829;
   1:L PR[91] R[100]mm/sec CNT100;
   1:  PR[GP1:91,1] = PR[GP1:90,1] + 48.522;
   1:  PR[GP1:91,2] = PR[GP1:90,2] + -11.612;
   1:L PR[91] R[100]mm/sec CNT100;
   1:  PR[GP1:91,1] = PR[GP1:90,1] + 50.130;
   1:  PR[GP1:91,2] = PR[GP1:90,2] + -0.085;
   1:L PR[91] R[100]mm/sec CNT100;
   1:  PR[GP1:91,1] = PR[GP1:90,1] + 49.730;
   1:  PR[GP1:91,2] = PR[GP1:90,2] + 2.101;
   1:L PR[91] R[100]mm/sec CNT100;
   1:  PR[GP1:91,1] = PR[GP1:90,1] + 48.113;
   1:  PR[GP1:91,2] = PR[GP1:90,2] + 13.697;
   1:L PR[91] R[100]mm/sec CNT100;
   1:  PR[GP1:91,1] = PR[GP1:90,1] + 43.405;
   1:  PR[GP1:91,2] = PR[GP1:90,2] + 24.360;
   1:L PR[91] R[100]mm/sec CNT100;
   1:  PR[GP1:91,1] = PR[GP1:90,1] + 42.268;
   1:  PR[GP1:91,2] = PR[GP1:90,2] + 26.259;
   1:L PR[91] R[100]mm/sec CNT100;
   1:  PR[GP1:91,1] = PR[GP1:90,1] + 34.779;
   1:  PR[GP1:91,2] = PR[GP1:90,2] + 35.281;
   1:L PR[91] R[100]mm/sec CNT100;
   1:  PR[GP1:91,1] = PR[GP1:90,1] + 33.110;
   1:  PR[GP1:91,2] = PR[GP1:90,2] + 36.620;
   1:L PR[91] R[100]mm/sec CNT100;
   1:  PR[GP1:91,1] = PR[GP1:90,1] + 24.533;
   1:  PR[GP1:91,2] = PR[GP1:90,2] + 42.693;
   1:L PR[91] R[100]mm/sec CNT100;
   1:  PR[GP1:91,1] = PR[GP1:90,1] + 14.729;
   1:  PR[GP1:91,2] = PR[GP1:90,2] + 46.492;
   1:L PR[91] R[100]mm/sec CNT100;
   1:  PR[GP1:91,1] = PR[GP1:90,1] + 12.735;
   1:  PR[GP1:91,2] = PR[GP1:90,2] + 47.163;
   1:L PR[91] R[100]mm/sec CNT100;
   1:  PR[GP1:91,1] = PR[GP1:90,1] + 2.237;
   1:  PR[GP1:91,2] = PR[GP1:90,2] + 48.463;
   1:L PR[91] R[100]mm/sec CNT100;
   1:  PR[GP1:91,1] = PR[GP1:90,1] + -0.013;
   1:  PR[GP1:91,2] = PR[GP1:90,2] + 48.420;
   1:L PR[91] R[100]mm/sec CNT100;
   1:  ! -- Layer/Ebene 205 -- !;
   1:  PR[91] = PR[90];
   1:  PR[GP1:91,1] = PR[GP1:90,1] + -1.657;
   1:  PR[GP1:91,2] = PR[GP1:90,2] + 48.611;
   1:  PR[GP1:91,3] = PR[GP1:90,3] + 125.355;
   1:L PR[91] R[100]mm/sec CNT100;
   1:  PR[GP1:91,1] = PR[GP1:90,1] + -12.427;
   1:  PR[GP1:91,2] = PR[GP1:90,2] + 47.277;
   1:L PR[91] R[100]mm/sec CNT100;
   1:  PR[GP1:91,1] = PR[GP1:90,1] + -14.068;
   1:  PR[GP1:91,2] = PR[GP1:90,2] + 46.725;
   1:L PR[91] R[100]mm/sec CNT100;
   1:  PR[GP1:91,1] = PR[GP1:90,1] + -24.123;
   1:  PR[GP1:91,2] = PR[GP1:90,2] + 42.828;
   1:L PR[91] R[100]mm/sec CNT100;
   1:  PR[GP1:91,1] = PR[GP1:90,1] + -25.546;
   1:  PR[GP1:91,2] = PR[GP1:90,2] + 41.691;
   1:L PR[91] R[100]mm/sec CNT100;
   1:  PR[GP1:91,1] = PR[GP1:90,1] + -34.335;
   1:  PR[GP1:91,2] = PR[GP1:90,2] + 35.468;
   1:L PR[91] R[100]mm/sec CNT100;
   1:  PR[GP1:91,1] = PR[GP1:90,1] + -42.031;
   1:  PR[GP1:91,2] = PR[GP1:90,2] + 26.198;
   1:L PR[91] R[100]mm/sec CNT100;
   1:  PR[GP1:91,1] = PR[GP1:90,1] + -42.966;
   1:  PR[GP1:91,2] = PR[GP1:90,2] + 24.636;
   1:L PR[91] R[100]mm/sec CNT100;
   1:  PR[GP1:91,1] = PR[GP1:90,1] + -47.820;
   1:  PR[GP1:91,2] = PR[GP1:90,2] + 13.641;
   1:L PR[91] R[100]mm/sec CNT100;
   1:  PR[GP1:91,1] = PR[GP1:90,1] + -48.152;
   1:  PR[GP1:91,2] = PR[GP1:90,2] + 11.819;
   1:L PR[91] R[100]mm/sec CNT100;
   1:  PR[GP1:91,1] = PR[GP1:90,1] + -49.809;
   1:  PR[GP1:91,2] = PR[GP1:90,2] + -0.059;
   1:L PR[91] R[100]mm/sec CNT100;
   1:  PR[GP1:91,1] = PR[GP1:90,1] + -49.480;
   1:  PR[GP1:91,2] = PR[GP1:90,2] + -1.856;
   1:L PR[91] R[100]mm/sec CNT100;
   1:  PR[GP1:91,1] = PR[GP1:90,1] + -47.814;
   1:  PR[GP1:91,2] = PR[GP1:90,2] + -13.797;
   1:L PR[91] R[100]mm/sec CNT100;
   1:  PR[GP1:91,1] = PR[GP1:90,1] + -42.966;
   1:  PR[GP1:91,2] = PR[GP1:90,2] + -24.780;
   1:L PR[91] R[100]mm/sec CNT100;
   1:  PR[GP1:91,1] = PR[GP1:90,1] + -42.031;
   1:  PR[GP1:91,2] = PR[GP1:90,2] + -26.342;
   1:L PR[91] R[100]mm/sec CNT100;
   1:  PR[GP1:91,1] = PR[GP1:90,1] + -34.324;
   1:  PR[GP1:91,2] = PR[GP1:90,2] + -35.625;
   1:L PR[91] R[100]mm/sec CNT100;
   1:  PR[GP1:91,1] = PR[GP1:90,1] + -32.952;
   1:  PR[GP1:91,2] = PR[GP1:90,2] + -36.726;
   1:L PR[91] R[100]mm/sec CNT100;
   1:  PR[GP1:91,1] = PR[GP1:90,1] + -24.140;
   1:  PR[GP1:91,2] = PR[GP1:90,2] + -42.966;
   1:L PR[91] R[100]mm/sec CNT100;
   1:  PR[GP1:91,1] = PR[GP1:90,1] + -14.068;
   1:  PR[GP1:91,2] = PR[GP1:90,2] + -46.869;
   1:L PR[91] R[100]mm/sec CNT100;
   1:  PR[GP1:91,1] = PR[GP1:90,1] + -12.428;
   1:  PR[GP1:91,2] = PR[GP1:90,2] + -47.421;
   1:L PR[91] R[100]mm/sec CNT100;
   1:  PR[GP1:91,1] = PR[GP1:90,1] + -1.657;
   1:  PR[GP1:91,2] = PR[GP1:90,2] + -48.755;
   1:L PR[91] R[100]mm/sec CNT100;
   1:  PR[GP1:91,1] = PR[GP1:90,1] + 0.007;
   1:  PR[GP1:91,2] = PR[GP1:90,2] + -48.720;
   1:L PR[91] R[100]mm/sec CNT100;
   1:  PR[GP1:91,1] = PR[GP1:90,1] + 1.867;
   1:  PR[GP1:91,2] = PR[GP1:90,2] + -48.755;
   1:L PR[91] R[100]mm/sec CNT100;
   1:  PR[GP1:91,1] = PR[GP1:90,1] + 12.639;
   1:  PR[GP1:91,2] = PR[GP1:90,2] + -47.421;
   1:L PR[91] R[100]mm/sec CNT100;
   1:  PR[GP1:91,1] = PR[GP1:90,1] + 14.280;
   1:  PR[GP1:91,2] = PR[GP1:90,2] + -46.869;
   1:L PR[91] R[100]mm/sec CNT100;
   1:  PR[GP1:91,1] = PR[GP1:90,1] + 24.336;
   1:  PR[GP1:91,2] = PR[GP1:90,2] + -42.972;
   1:L PR[91] R[100]mm/sec CNT100;
   1:  PR[GP1:91,1] = PR[GP1:90,1] + 25.759;
   1:  PR[GP1:91,2] = PR[GP1:90,2] + -41.835;
   1:L PR[91] R[100]mm/sec CNT100;
   1:  PR[GP1:91,1] = PR[GP1:90,1] + 34.550;
   1:  PR[GP1:91,2] = PR[GP1:90,2] + -35.610;
   1:L PR[91] R[100]mm/sec CNT100;
   1:  PR[GP1:91,1] = PR[GP1:90,1] + 42.245;
   1:  PR[GP1:91,2] = PR[GP1:90,2] + -26.341;
   1:L PR[91] R[100]mm/sec CNT100;
   1:  PR[GP1:91,1] = PR[GP1:90,1] + 43.179;
   1:  PR[GP1:91,2] = PR[GP1:90,2] + -24.780;
   1:L PR[91] R[100]mm/sec CNT100;
   1:  PR[GP1:91,1] = PR[GP1:90,1] + 48.033;
   1:  PR[GP1:91,2] = PR[GP1:90,2] + -13.785;
   1:L PR[91] R[100]mm/sec CNT100;
   1:  PR[GP1:91,1] = PR[GP1:90,1] + 48.365;
   1:  PR[GP1:91,2] = PR[GP1:90,2] + -11.962;
   1:L PR[91] R[100]mm/sec CNT100;
   1:  PR[GP1:91,1] = PR[GP1:90,1] + 50.022;
   1:  PR[GP1:91,2] = PR[GP1:90,2] + -0.085;
   1:L PR[91] R[100]mm/sec CNT100;
   1:  PR[GP1:91,1] = PR[GP1:90,1] + 49.693;
   1:  PR[GP1:91,2] = PR[GP1:90,2] + 1.713;
   1:L PR[91] R[100]mm/sec CNT100;
   1:  PR[GP1:91,1] = PR[GP1:90,1] + 48.028;
   1:  PR[GP1:91,2] = PR[GP1:90,2] + 13.653;
   1:L PR[91] R[100]mm/sec CNT100;
   1:  PR[GP1:91,1] = PR[GP1:90,1] + 43.179;
   1:  PR[GP1:91,2] = PR[GP1:90,2] + 24.636;
   1:L PR[91] R[100]mm/sec CNT100;
   1:  PR[GP1:91,1] = PR[GP1:90,1] + 42.245;
   1:  PR[GP1:91,2] = PR[GP1:90,2] + 26.197;
   1:L PR[91] R[100]mm/sec CNT100;
   1:  PR[GP1:91,1] = PR[GP1:90,1] + 34.538;
   1:  PR[GP1:91,2] = PR[GP1:90,2] + 35.480;
   1:L PR[91] R[100]mm/sec CNT100;
   1:  PR[GP1:91,1] = PR[GP1:90,1] + 33.166;
   1:  PR[GP1:91,2] = PR[GP1:90,2] + 36.581;
   1:L PR[91] R[100]mm/sec CNT100;
   1:  PR[GP1:91,1] = PR[GP1:90,1] + 24.353;
   1:  PR[GP1:91,2] = PR[GP1:90,2] + 42.822;
   1:L PR[91] R[100]mm/sec CNT100;
   1:  PR[GP1:91,1] = PR[GP1:90,1] + 14.279;
   1:  PR[GP1:91,2] = PR[GP1:90,2] + 46.725;
   1:L PR[91] R[100]mm/sec CNT100;
   1:  PR[GP1:91,1] = PR[GP1:90,1] + 12.639;
   1:  PR[GP1:91,2] = PR[GP1:90,2] + 47.277;
   1:L PR[91] R[100]mm/sec CNT100;
   1:  PR[GP1:91,1] = PR[GP1:90,1] + 1.866;
   1:  PR[GP1:91,2] = PR[GP1:90,2] + 48.611;
   1:L PR[91] R[100]mm/sec CNT100;
   1:  PR[GP1:91,1] = PR[GP1:90,1] + 0.007;
   1:  PR[GP1:91,2] = PR[GP1:90,2] + 48.576;
   1:L PR[91] R[100]mm/sec CNT100;
   1:  ! -- Layer/Ebene 206 -- !;
   1:  PR[91] = PR[90];
   1:  PR[GP1:91,1] = PR[GP1:90,1] + -1.286;
   1:  PR[GP1:91,2] = PR[GP1:90,2] + 48.759;
   1:  PR[GP1:91,3] = PR[GP1:90,3] + 125.965;
   1:L PR[91] R[100]mm/sec CNT100;
   1:  PR[GP1:91,1] = PR[GP1:90,1] + -12.331;
   1:  PR[GP1:91,2] = PR[GP1:90,2] + 47.391;
   1:L PR[91] R[100]mm/sec CNT100;
   1:  PR[GP1:91,1] = PR[GP1:90,1] + -13.617;
   1:  PR[GP1:91,2] = PR[GP1:90,2] + 46.958;
   1:L PR[91] R[100]mm/sec CNT100;
   1:  PR[GP1:91,1] = PR[GP1:90,1] + -23.943;
   1:  PR[GP1:91,2] = PR[GP1:90,2] + 42.957;
   1:L PR[91] R[100]mm/sec CNT100;
   1:  PR[GP1:91,1] = PR[GP1:90,1] + -25.060;
   1:  PR[GP1:91,2] = PR[GP1:90,2] + 42.064;
   1:L PR[91] R[100]mm/sec CNT100;
   1:  PR[GP1:91,1] = PR[GP1:90,1] + -34.094;
   1:  PR[GP1:91,2] = PR[GP1:90,2] + 35.667;
   1:L PR[91] R[100]mm/sec CNT100;
   1:  PR[GP1:91,1] = PR[GP1:90,1] + -42.007;
   1:  PR[GP1:91,2] = PR[GP1:90,2] + 26.136;
   1:L PR[91] R[100]mm/sec CNT100;
   1:  PR[GP1:91,1] = PR[GP1:90,1] + -42.740;
   1:  PR[GP1:91,2] = PR[GP1:90,2] + 24.912;
   1:L PR[91] R[100]mm/sec CNT100;
   1:  PR[GP1:91,1] = PR[GP1:90,1] + -47.734;
   1:  PR[GP1:91,2] = PR[GP1:90,2] + 13.598;
   1:L PR[91] R[100]mm/sec CNT100;
   1:  PR[GP1:91,1] = PR[GP1:90,1] + -47.995;
   1:  PR[GP1:91,2] = PR[GP1:90,2] + 12.169;
   1:L PR[91] R[100]mm/sec CNT100;
   1:  PR[GP1:91,1] = PR[GP1:90,1] + -49.700;
   1:  PR[GP1:91,2] = PR[GP1:90,2] + -0.059;
   1:L PR[91] R[100]mm/sec CNT100;
   1:  PR[GP1:91,1] = PR[GP1:90,1] + -49.443;
   1:  PR[GP1:91,2] = PR[GP1:90,2] + -1.467;
   1:L PR[91] R[100]mm/sec CNT100;
   1:  PR[GP1:91,1] = PR[GP1:90,1] + -47.729;
   1:  PR[GP1:91,2] = PR[GP1:90,2] + -13.754;
   1:L PR[91] R[100]mm/sec CNT100;
   1:  PR[GP1:91,1] = PR[GP1:90,1] + -42.740;
   1:  PR[GP1:91,2] = PR[GP1:90,2] + -25.056;
   1:L PR[91] R[100]mm/sec CNT100;
   1:  PR[GP1:91,1] = PR[GP1:90,1] + -42.007;
   1:  PR[GP1:91,2] = PR[GP1:90,2] + -26.280;
   1:L PR[91] R[100]mm/sec CNT100;
   1:  PR[GP1:91,1] = PR[GP1:90,1] + -34.083;
   1:  PR[GP1:91,2] = PR[GP1:90,2] + -35.824;
   1:L PR[91] R[100]mm/sec CNT100;
   1:  PR[GP1:91,1] = PR[GP1:90,1] + -33.008;
   1:  PR[GP1:91,2] = PR[GP1:90,2] + -36.687;
   1:L PR[91] R[100]mm/sec CNT100;
   1:  PR[GP1:91,1] = PR[GP1:90,1] + -23.959;
   1:  PR[GP1:91,2] = PR[GP1:90,2] + -43.094;
   1:L PR[91] R[100]mm/sec CNT100;
   1:  PR[GP1:91,1] = PR[GP1:90,1] + -13.617;
   1:  PR[GP1:91,2] = PR[GP1:90,2] + -47.102;
   1:L PR[91] R[100]mm/sec CNT100;
   1:  PR[GP1:91,1] = PR[GP1:90,1] + -12.331;
   1:  PR[GP1:91,2] = PR[GP1:90,2] + -47.535;
   1:L PR[91] R[100]mm/sec CNT100;
   1:  PR[GP1:91,1] = PR[GP1:90,1] + -1.287;
   1:  PR[GP1:91,2] = PR[GP1:90,2] + -48.903;
   1:L PR[91] R[100]mm/sec CNT100;
   1:  PR[GP1:91,1] = PR[GP1:90,1] + 0.027;
   1:  PR[GP1:91,2] = PR[GP1:90,2] + -48.875;
   1:L PR[91] R[100]mm/sec CNT100;
   1:  PR[GP1:91,1] = PR[GP1:90,1] + 1.496;
   1:  PR[GP1:91,2] = PR[GP1:90,2] + -48.903;
   1:L PR[91] R[100]mm/sec CNT100;
   1:  PR[GP1:91,1] = PR[GP1:90,1] + 12.542;
   1:  PR[GP1:91,2] = PR[GP1:90,2] + -47.535;
   1:L PR[91] R[100]mm/sec CNT100;
   1:  PR[GP1:91,1] = PR[GP1:90,1] + 13.829;
   1:  PR[GP1:91,2] = PR[GP1:90,2] + -47.102;
   1:L PR[91] R[100]mm/sec CNT100;
   1:  PR[GP1:91,1] = PR[GP1:90,1] + 24.156;
   1:  PR[GP1:91,2] = PR[GP1:90,2] + -43.101;
   1:L PR[91] R[100]mm/sec CNT100;
   1:  PR[GP1:91,1] = PR[GP1:90,1] + 25.273;
   1:  PR[GP1:91,2] = PR[GP1:90,2] + -42.208;
   1:L PR[91] R[100]mm/sec CNT100;
   1:  PR[GP1:91,1] = PR[GP1:90,1] + 34.310;
   1:  PR[GP1:91,2] = PR[GP1:90,2] + -35.809;
   1:L PR[91] R[100]mm/sec CNT100;
   1:  PR[GP1:91,1] = PR[GP1:90,1] + 42.221;
   1:  PR[GP1:91,2] = PR[GP1:90,2] + -26.279;
   1:L PR[91] R[100]mm/sec CNT100;
   1:  PR[GP1:91,1] = PR[GP1:90,1] + 42.953;
   1:  PR[GP1:91,2] = PR[GP1:90,2] + -25.055;
   1:L PR[91] R[100]mm/sec CNT100;
   1:  PR[GP1:91,1] = PR[GP1:90,1] + 47.948;
   1:  PR[GP1:91,2] = PR[GP1:90,2] + -13.742;
   1:L PR[91] R[100]mm/sec CNT100;
   1:  PR[GP1:91,1] = PR[GP1:90,1] + 48.208;
   1:  PR[GP1:91,2] = PR[GP1:90,2] + -12.313;
   1:L PR[91] R[100]mm/sec CNT100;
   1:  PR[GP1:91,1] = PR[GP1:90,1] + 49.914;
   1:  PR[GP1:91,2] = PR[GP1:90,2] + -0.085;
   1:L PR[91] R[100]mm/sec CNT100;
   1:  PR[GP1:91,1] = PR[GP1:90,1] + 49.656;
   1:  PR[GP1:91,2] = PR[GP1:90,2] + 1.324;
   1:L PR[91] R[100]mm/sec CNT100;
   1:  PR[GP1:91,1] = PR[GP1:90,1] + 47.943;
   1:  PR[GP1:91,2] = PR[GP1:90,2] + 13.610;
   1:L PR[91] R[100]mm/sec CNT100;
   1:  PR[GP1:91,1] = PR[GP1:90,1] + 42.953;
   1:  PR[GP1:91,2] = PR[GP1:90,2] + 24.911;
   1:L PR[91] R[100]mm/sec CNT100;
   1:  PR[GP1:91,1] = PR[GP1:90,1] + 42.221;
   1:  PR[GP1:91,2] = PR[GP1:90,2] + 26.135;
   1:L PR[91] R[100]mm/sec CNT100;
   1:  PR[GP1:91,1] = PR[GP1:90,1] + 34.298;
   1:  PR[GP1:91,2] = PR[GP1:90,2] + 35.679;
   1:L PR[91] R[100]mm/sec CNT100;
   1:  PR[GP1:91,1] = PR[GP1:90,1] + 33.222;
   1:  PR[GP1:91,2] = PR[GP1:90,2] + 36.542;
   1:L PR[91] R[100]mm/sec CNT100;
   1:  PR[GP1:91,1] = PR[GP1:90,1] + 24.172;
   1:  PR[GP1:91,2] = PR[GP1:90,2] + 42.950;
   1:L PR[91] R[100]mm/sec CNT100;
   1:  PR[GP1:91,1] = PR[GP1:90,1] + 13.829;
   1:  PR[GP1:91,2] = PR[GP1:90,2] + 46.959;
   1:L PR[91] R[100]mm/sec CNT100;
   1:  PR[GP1:91,1] = PR[GP1:90,1] + 12.542;
   1:  PR[GP1:91,2] = PR[GP1:90,2] + 47.392;
   1:L PR[91] R[100]mm/sec CNT100;
   1:  PR[GP1:91,1] = PR[GP1:90,1] + 1.495;
   1:  PR[GP1:91,2] = PR[GP1:90,2] + 48.759;
   1:L PR[91] R[100]mm/sec CNT100;
   1:  PR[GP1:91,1] = PR[GP1:90,1] + 0.027;
   1:  PR[GP1:91,2] = PR[GP1:90,2] + 48.731;
   1:L PR[91] R[100]mm/sec CNT100 TB   .50sec,CALL END_PUD;
   1:  DO[117:Laser Start]=OFF;
   1:  !Sicherheitspunkt!;
   1:  PR[92] = PR[91];
   1:  PR[92] = PR[GP1:92,3] + 50;
   1:J PR[92];
   1:  WAIT   5.00(sec);
   1:  DO[119:Gas]=OFF;
   1:  CALL HOME_ALL;
/POS
/END
